C05481=1226.735,157.373,-52.424,-177.853,5.794,148.385
C05482=1226.731,157.623,-52.446,-177.851,5.795,148.384
C05483=1226.726,157.871,-52.468,-177.848,5.797,148.384
C05484=1226.721,158.120,-52.490,-177.846,5.798,148.383
C05485=1226.717,158.370,-52.511,-177.843,5.799,148.383
C05486=1226.712,158.619,-52.533,-177.841,5.800,148.382
C05487=1226.707,158.867,-52.555,-177.838,5.802,148.382
C05488=1226.703,159.117,-52.577,-177.836,5.803,148.381
C05489=1226.697,159.386,-52.600,-177.833,5.804,148.381
C05490=1226.693,159.655,-52.623,-177.830,5.806,148.380
C05491=1226.687,159.924,-52.647,-177.828,5.807,148.380
C05492=1226.683,160.193,-52.670,-177.824,5.808,148.379
C05493=1226.678,160.441,-52.691,-177.822,5.810,148.379
C05494=1226.674,160.691,-52.713,-177.820,5.811,148.379
C05495=1226.669,160.939,-52.735,-177.817,5.813,148.378
C05496=1226.664,161.189,-52.756,-177.814,5.814,148.378
C05497=1226.659,161.438,-52.778,-177.812,5.815,148.377
C05498=1226.654,161.687,-52.800,-177.809,5.816,148.377
C05499=1226.649,161.936,-52.822,-177.807,5.818,148.376
C05500=1226.644,162.185,-52.844,-177.804,5.819,148.376
C05501=1226.640,162.434,-52.866,-177.801,5.820,148.375
C05502=1226.635,162.683,-52.888,-177.799,5.821,148.375
C05503=1226.630,162.932,-52.909,-177.797,5.823,148.375
C05504=1226.626,163.181,-52.931,-177.794,5.824,148.374
C05505=1226.621,163.430,-52.953,-177.791,5.826,148.374
C05506=1226.617,163.679,-52.975,-177.789,5.828,148.373
C05507=1226.612,163.928,-52.997,-177.786,5.828,148.373
C05508=1226.608,164.177,-53.019,-177.783,5.830,148.372
C05509=1226.603,164.426,-53.040,-177.781,5.831,148.372
C05510=1226.599,164.675,-53.062,-177.778,5.833,148.371
C05511=1226.594,164.924,-53.084,-177.776,5.834,148.371
C05512=1226.590,165.173,-53.106,-177.773,5.835,148.370
C05513=1226.584,165.422,-53.129,-177.771,5.836,148.370
C05514=1226.579,165.670,-53.150,-177.768,5.838,148.369
C05515=1226.575,165.920,-53.172,-177.766,5.839,148.369
C05516=1226.570,166.168,-53.194,-177.763,5.840,148.368
C05517=1226.566,166.418,-53.216,-177.760,5.842,148.368
C05518=1226.561,166.666,-53.238,-177.758,5.843,148.368
C05519=1226.557,166.916,-53.260,-177.755,5.845,148.367
C05520=1226.551,167.165,-53.282,-177.753,5.846,148.367
C05521=1226.547,167.414,-53.304,-177.750,5.848,148.366
C05522=1226.542,167.663,-53.326,-177.748,5.848,148.366
C05523=1226.538,167.912,-53.348,-177.745,5.850,148.365
C05524=1226.534,168.161,-53.371,-177.742,5.852,148.365
C05525=1226.528,168.410,-53.393,-177.740,5.853,148.365
C05526=1226.524,168.659,-53.415,-177.737,5.854,148.364
C05527=1226.519,168.908,-53.437,-177.735,5.855,148.364
C05528=1226.515,169.157,-53.459,-177.732,5.857,148.363
C05529=1226.510,169.406,-53.480,-177.730,5.858,148.363
C05530=1226.505,169.655,-53.504,-177.727,5.860,148.362
C05531=1226.500,169.903,-53.525,-177.724,5.861,148.362
C05532=1226.496,170.153,-53.547,-177.722,5.862,148.361
C05533=1226.490,170.402,-53.570,-177.719,5.864,148.361
C05534=1226.486,170.651,-53.592,-177.717,5.865,148.361
C05535=1226.482,170.899,-53.614,-177.715,5.867,148.360
C05536=1226.477,171.148,-53.636,-177.712,5.867,148.360
C05537=1226.472,171.398,-53.659,-177.709,5.869,148.359
C05538=1226.467,171.647,-53.681,-177.707,5.871,148.359
C05539=1226.463,171.895,-53.703,-177.704,5.872,148.358
C05540=1226.458,172.144,-53.726,-177.701,5.874,148.358
C05541=1226.454,172.394,-53.748,-177.699,5.875,148.358
C05542=1226.449,172.642,-53.770,-177.697,5.876,148.357
C05543=1226.444,172.891,-53.793,-177.693,5.878,148.357
C05544=1226.440,173.141,-53.815,-177.691,5.879,148.356
C05545=1226.435,173.389,-53.837,-177.689,5.881,148.356
C05546=1226.430,173.638,-53.860,-177.687,5.882,148.356
C05547=1226.425,173.887,-53.881,-177.684,5.883,148.355
C05548=1226.421,174.136,-53.904,-177.681,5.885,148.355
C05549=1226.416,174.385,-53.927,-177.679,5.886,148.354
C05550=1226.412,174.633,-53.949,-177.676,5.888,148.354
C05551=1226.407,174.883,-53.971,-177.674,5.889,148.353
C05552=1226.402,175.132,-53.994,-177.671,5.890,148.353
C05553=1226.398,175.380,-54.016,-177.668,5.892,148.353
C05554=1226.393,175.630,-54.039,-177.666,5.893,148.352
C05555=1226.389,175.879,-54.062,-177.663,5.895,148.352
C05556=1226.384,176.127,-54.083,-177.660,5.897,148.351
C05557=1226.379,176.376,-54.107,-177.658,5.898,148.351
C05558=1226.375,176.626,-54.129,-177.655,5.899,148.350
C05559=1226.370,176.874,-54.152,-177.653,5.900,148.350
C05560=1226.366,177.123,-54.174,-177.650,5.902,148.349
C05561=1226.361,177.372,-54.197,-177.648,5.904,148.349
C05562=1226.356,177.621,-54.219,-177.645,5.905,148.349
C05563=1226.352,177.870,-54.242,-177.642,5.906,148.348
C05564=1226.347,178.119,-54.264,-177.640,5.908,148.348
C05565=1226.342,178.367,-54.287,-177.638,5.909,148.347
C05566=1226.337,178.617,-54.309,-177.635,5.911,148.347
C05567=1226.333,178.866,-54.332,-177.633,5.912,148.346
C05568=1226.328,179.115,-54.354,-177.630,5.914,148.346
C05569=1226.324,179.364,-54.377,-177.627,5.915,148.346
C05570=1226.319,179.613,-54.401,-177.625,5.916,148.345
C05571=1226.315,179.862,-54.423,-177.622,5.918,148.345
C05572=1226.310,180.110,-54.446,-177.619,5.920,148.344
C05573=1226.305,180.360,-54.468,-177.617,5.921,148.344
C05574=1226.301,180.609,-54.491,-177.615,5.923,148.344
C05575=1226.295,180.857,-54.514,-177.611,5.924,148.343
C05576=1226.291,181.106,-54.536,-177.609,5.925,148.343
C05577=1226.286,181.355,-54.559,-177.607,5.927,148.342
C05578=1226.282,181.604,-54.582,-177.604,5.929,148.342
C05579=1226.277,181.853,-54.604,-177.601,5.929,148.341
C05580=1226.273,182.102,-54.627,-177.599,5.931,148.341
C05581=1226.268,182.351,-54.651,-177.596,5.933,148.341
C05582=1226.263,182.600,-54.674,-177.594,5.934,148.340
C05583=1226.259,182.848,-54.696,-177.591,5.936,148.340
C05584=1226.254,183.097,-54.719,-177.589,5.937,148.339
C05585=1226.250,183.346,-54.742,-177.586,5.938,148.339
C05586=1226.245,183.595,-54.765,-177.584,5.940,148.339
C05587=1226.240,183.845,-54.788,-177.581,5.941,148.338
C05588=1226.236,184.093,-54.810,-177.578,5.943,148.338
C05589=1226.231,184.342,-54.833,-177.576,5.945,148.337
C05590=1226.226,184.591,-54.857,-177.574,5.946,148.337
C05591=1226.222,184.840,-54.880,-177.571,5.947,148.337
C05592=1226.217,185.089,-54.902,-177.568,5.949,148.336
C05593=1226.213,185.359,-54.927,-177.565,5.951,148.336
C05594=1226.208,185.628,-54.952,-177.563,5.953,148.335
C05595=1226.202,185.898,-54.977,-177.560,5.955,148.335
C05596=1226.198,186.167,-55.002,-177.557,5.955,148.334
C05597=1226.193,186.416,-55.025,-177.555,5.957,148.334
C05598=1226.187,186.665,-55.048,-177.552,5.959,148.334
C05599=1226.183,186.914,-55.071,-177.549,5.961,148.333
C05600=1226.179,187.163,-55.094,-177.547,5.961,148.333
C05601=1226.174,187.412,-55.117,-177.544,5.963,148.332
C05602=1226.169,187.661,-55.140,-177.542,5.965,148.332
C05603=1226.165,187.910,-55.163,-177.539,5.966,148.332
C05604=1226.161,188.159,-55.187,-177.537,5.968,148.331
C05605=1226.155,188.407,-55.210,-177.534,5.969,148.331
C05606=1226.151,188.656,-55.233,-177.532,5.970,148.330
C05607=1226.146,188.905,-55.256,-177.529,5.972,148.330
C05608=1226.142,189.154,-55.279,-177.526,5.974,148.330
C05609=1226.137,189.403,-55.302,-177.524,5.975,148.329
C05610=1226.133,189.652,-55.326,-177.522,5.977,148.329
C05611=1226.128,189.901,-55.349,-177.518,5.979,148.328
C05612=1226.124,190.150,-55.372,-177.516,5.980,148.328
C05613=1226.119,190.398,-55.395,-177.514,5.981,148.328
C05614=1226.114,190.647,-55.418,-177.511,5.983,148.327
C05615=1226.109,190.896,-55.442,-177.508,5.985,148.327
C05616=1226.105,191.145,-55.465,-177.506,5.986,148.327
C05617=1226.100,191.394,-55.488,-177.503,5.988,148.326
C05618=1226.096,191.643,-55.511,-177.501,5.989,148.326
C05619=1226.092,191.891,-55.535,-177.498,5.991,148.325
C05620=1226.087,192.140,-55.558,-177.496,5.992,148.325
C05621=1226.082,192.389,-55.582,-177.493,5.994,148.325
C05622=1226.077,192.638,-55.605,-177.491,5.996,148.324
C05623=1226.073,192.887,-55.629,-177.487,5.997,148.324
C05624=1226.068,193.136,-55.652,-177.485,5.999,148.323
C05625=1226.063,193.385,-55.675,-177.483,6.000,148.323
C05626=1226.060,193.634,-55.699,-177.480,6.002,148.323
C05627=1226.054,193.882,-55.722,-177.478,6.003,148.322
C05628=1226.050,194.131,-55.745,-177.475,6.005,148.322
C05629=1226.045,194.380,-55.768,-177.473,6.007,148.322
C05630=1226.040,194.629,-55.792,-177.470,6.008,148.321
C05631=1226.036,194.877,-55.816,-177.467,6.009,148.321
C05632=1226.031,195.126,-55.839,-177.465,6.011,148.320
C05633=1226.027,195.375,-55.863,-177.462,6.013,148.320
C05634=1226.022,195.624,-55.886,-177.460,6.015,148.320
C05635=1226.017,195.873,-55.910,-177.457,6.016,148.319
C05636=1226.013,196.122,-55.933,-177.455,6.018,148.319
C05637=1226.008,196.371,-55.957,-177.452,6.019,148.318
C05638=1226.003,196.620,-55.980,-177.449,6.021,148.318
C05639=1225.999,196.868,-56.004,-177.447,6.022,148.318
C05640=1225.994,197.117,-56.028,-177.444,6.024,148.317
C05641=1225.990,197.366,-56.051,-177.442,6.026,148.317
C05642=1225.985,197.615,-56.075,-177.439,6.028,148.317
C05643=1225.980,197.864,-56.098,-177.437,6.029,148.316
C05644=1225.976,198.113,-56.122,-177.434,6.031,148.316
C05645=1225.971,198.361,-56.146,-177.431,6.032,148.315
C05646=1225.967,198.610,-56.169,-177.429,6.034,148.315
C05647=1225.963,198.859,-56.194,-177.426,6.035,148.315
C05648=1225.958,199.109,-56.217,-177.424,6.037,148.314
C05649=1225.953,199.358,-56.240,-177.421,6.039,148.314
C05650=1225.949,199.606,-56.264,-177.419,6.041,148.313
C05651=1225.944,199.855,-56.288,-177.416,6.042,148.313
C05652=1225.940,200.103,-56.312,-177.414,6.043,148.313
C05653=1225.935,200.352,-56.335,-177.411,6.045,148.312
C05654=1225.930,200.601,-56.360,-177.408,6.047,148.312
C05655=1225.925,200.850,-56.383,-177.405,6.049,148.312
C05656=1225.921,201.099,-56.407,-177.403,6.050,148.311
C05657=1225.916,201.348,-56.431,-177.401,6.052,148.311
C05658=1225.912,201.596,-56.455,-177.398,6.053,148.310
C05659=1225.907,201.845,-56.478,-177.395,6.055,148.310
C05660=1225.903,202.094,-56.502,-177.393,6.057,148.310
C05661=1225.899,202.343,-56.526,-177.391,6.058,148.309
C05662=1225.894,202.592,-56.551,-177.388,6.060,148.309
C05663=1225.889,202.841,-56.574,-177.385,6.062,148.309
C05664=1225.885,203.089,-56.598,-177.383,6.064,148.308
C05665=1225.880,203.338,-56.622,-177.380,6.064,148.308
C05666=1225.875,203.587,-56.645,-177.378,6.066,148.307
C05667=1225.871,203.835,-56.669,-177.375,6.068,148.307
C05668=1225.866,204.085,-56.694,-177.372,6.070,148.307
C05669=1225.862,204.334,-56.718,-177.370,6.072,148.306
C05670=1225.857,204.582,-56.742,-177.368,6.073,148.306
C05671=1225.853,204.831,-56.765,-177.365,6.075,148.306
C05672=1225.848,205.080,-56.789,-177.362,6.076,148.305
C05673=1225.843,205.328,-56.814,-177.360,6.078,148.305
C05674=1225.839,205.577,-56.837,-177.357,6.080,148.305
C05675=1225.835,205.826,-56.862,-177.354,6.082,148.304
C05676=1225.830,206.075,-56.886,-177.352,6.083,148.304
C05677=1225.825,206.324,-56.910,-177.349,6.085,148.303
C05678=1225.820,206.573,-56.934,-177.347,6.086,148.303
C05679=1225.816,206.821,-56.958,-177.344,6.088,148.303
C05680=1225.812,207.070,-56.982,-177.341,6.090,148.302
C05681=1225.807,207.319,-57.006,-177.339,6.091,148.302
C05682=1225.802,207.568,-57.030,-177.337,6.093,148.302
C05683=1225.798,207.816,-57.055,-177.334,6.095,148.301
C05684=1225.793,208.065,-57.079,-177.331,6.097,148.301
C05685=1225.789,208.315,-57.103,-177.329,6.099,148.301
C05686=1225.784,208.563,-57.127,-177.326,6.100,148.300
C05687=1225.779,208.812,-57.152,-177.324,6.101,148.300
C05688=1225.775,209.060,-57.176,-177.321,6.103,148.300
C05689=1225.771,209.309,-57.200,-177.319,6.105,148.299
C05690=1225.766,209.558,-57.225,-177.316,6.107,148.299
C05691=1225.761,209.807,-57.248,-177.313,6.109,148.299
C05692=1225.757,210.056,-57.272,-177.311,6.111,148.298
C05693=1225.752,210.304,-57.297,-177.309,6.112,148.298
C05694=1225.748,210.553,-57.321,-177.306,6.114,148.298
C05695=1225.743,210.802,-57.346,-177.303,6.115,148.297
C05696=1225.738,211.051,-57.370,-177.300,6.117,148.297
C05697=1225.733,211.321,-57.397,-177.298,6.119,148.296
C05698=1225.728,211.592,-57.423,-177.295,6.121,148.296
C05699=1225.724,211.862,-57.449,-177.292,6.123,148.296
C05700=1225.719,212.132,-57.476,-177.290,6.124,148.295
C05701=1225.714,212.381,-57.501,-177.287,6.126,148.295
C05702=1225.710,212.630,-57.525,-177.285,6.128,148.295
C05703=1225.705,212.879,-57.550,-177.281,6.130,148.294
C05704=1225.700,213.127,-57.574,-177.279,6.132,148.294
C05705=1225.696,213.376,-57.598,-177.276,6.133,148.294
C05706=1225.692,213.625,-57.623,-177.274,6.135,148.293
C05707=1225.687,213.873,-57.647,-177.271,6.136,148.293
C05708=1225.682,214.122,-57.672,-177.269,6.138,148.293
C05709=1225.678,214.371,-57.696,-177.266,6.140,148.292
C05710=1225.673,214.620,-57.721,-177.264,6.142,148.292
C05711=1225.669,214.868,-57.745,-177.261,6.144,148.292
C05712=1225.664,215.118,-57.770,-177.258,6.146,148.291
C05713=1225.660,215.366,-57.794,-177.256,6.147,148.291
C05714=1225.655,215.615,-57.819,-177.254,6.148,148.290
C05715=1225.651,215.863,-57.844,-177.251,6.150,148.290
C05716=1225.646,216.112,-57.869,-177.248,6.152,148.290
C05717=1225.641,216.361,-57.893,-177.246,6.154,148.289
C05718=1225.637,216.610,-57.918,-177.243,6.156,148.289
C05719=1225.632,216.859,-57.942,-177.240,6.158,148.289
C05720=1225.628,217.108,-57.967,-177.238,6.160,148.289
C05721=1225.623,217.356,-57.992,-177.235,6.161,148.288
C05722=1225.619,217.604,-58.016,-177.233,6.163,148.288
C05723=1225.614,217.854,-58.041,-177.230,6.164,148.287
C05724=1225.609,218.103,-58.066,-177.228,6.166,148.287
C05725=1225.605,218.351,-58.090,-177.225,6.168,148.287
C05726=1225.601,218.600,-58.116,-177.223,6.170,148.286
C05727=1225.596,218.848,-58.140,-177.220,6.172,148.286
C05728=1225.592,219.098,-58.165,-177.217,6.174,148.286
C05729=1225.587,219.346,-58.190,-177.215,6.175,148.286
C05730=1225.582,219.594,-58.214,-177.212,6.177,148.285
C05731=1225.578,219.844,-58.239,-177.209,6.179,148.285
C05732=1225.573,220.092,-58.264,-177.207,6.180,148.284
C05733=1225.569,220.341,-58.289,-177.205,6.182,148.284
C05734=1225.564,220.589,-58.314,-177.202,6.184,148.284
C05735=1225.560,220.839,-58.339,-177.200,6.186,148.284
C05736=1225.556,221.087,-58.364,-177.197,6.188,148.283
C05737=1225.550,221.335,-58.388,-177.195,6.190,148.283
C05738=1225.546,221.585,-58.413,-177.192,6.192,148.283
C05739=1225.542,221.833,-58.438,-177.189,6.194,148.282
C05740=1225.537,222.082,-58.463,-177.187,6.195,148.282
C05741=1225.532,222.330,-58.489,-177.184,6.197,148.282
C05742=1225.529,222.579,-58.513,-177.182,6.198,148.281
C05743=1225.524,222.828,-58.538,-177.180,6.200,148.281
C05744=1225.519,223.077,-58.563,-177.177,6.202,148.281
C05745=1225.514,223.326,-58.588,-177.174,6.204,148.280
C05746=1225.511,223.574,-58.613,-177.172,6.206,148.280
C05747=1225.506,223.823,-58.638,-177.169,6.208,148.280
C05748=1225.501,224.072,-58.664,-177.166,6.210,148.279
C05749=1225.496,224.320,-58.688,-177.164,6.211,148.279
C05750=1225.492,224.569,-58.714,-177.161,6.213,148.279
C05751=1225.488,224.817,-58.738,-177.159,6.215,148.278
C05752=1225.483,225.066,-58.764,-177.156,6.217,148.278
C05753=1225.478,225.315,-58.789,-177.153,6.219,148.278
C05754=1225.474,225.564,-58.814,-177.151,6.220,148.277
C05755=1225.469,225.813,-58.839,-177.149,6.222,148.277
C05756=1225.465,226.061,-58.864,-177.146,6.224,148.277
C05757=1225.460,226.310,-58.889,-177.144,6.226,148.277
C05758=1225.456,226.559,-58.915,-177.141,6.228,148.276
C05759=1225.451,226.807,-58.940,-177.139,6.230,148.276
C05760=1225.447,227.056,-58.965,-177.136,6.231,148.276
C05761=1225.442,227.304,-58.990,-177.133,6.233,148.275
C05762=1225.438,227.553,-59.015,-177.131,6.235,148.275
C05763=1225.434,227.802,-59.041,-177.128,6.237,148.275
C05764=1225.429,228.050,-59.066,-177.125,6.239,148.274
C05765=1225.424,228.300,-59.091,-177.123,6.241,148.274
C05766=1225.420,228.548,-59.116,-177.120,6.243,148.274
C05767=1225.415,228.797,-59.142,-177.118,6.244,148.273
C05768=1225.410,229.045,-59.167,-177.116,6.246,148.273
C05769=1225.406,229.294,-59.193,-177.113,6.248,148.273
C05770=1225.402,229.543,-59.218,-177.111,6.250,148.273
C05771=1225.397,229.791,-59.244,-177.108,6.251,148.272
C05772=1225.393,230.040,-59.269,-177.105,6.253,148.272
C05773=1225.388,230.289,-59.294,-177.103,6.255,148.272
C05774=1225.384,230.537,-59.319,-177.100,6.257,148.271
C05775=1225.380,230.786,-59.345,-177.098,6.259,148.271
C05776=1225.375,231.035,-59.370,-177.095,6.261,148.271
C05777=1225.371,231.283,-59.395,-177.093,6.263,148.271
C05778=1225.366,231.531,-59.421,-177.090,6.265,148.270
C05779=1225.362,231.780,-59.447,-177.088,6.267,148.270
C05780=1225.357,232.029,-59.472,-177.085,6.269,148.270
C05781=1225.352,232.278,-59.497,-177.082,6.270,148.269
C05782=1225.348,232.527,-59.523,-177.080,6.272,148.269
C05783=1225.344,232.775,-59.549,-177.077,6.274,148.269
C05784=1225.339,233.024,-59.574,-177.075,6.276,148.268
C05785=1225.334,233.273,-59.600,-177.073,6.277,148.268
C05786=1225.330,233.521,-59.626,-177.070,6.279,148.268
C05787=1225.325,233.770,-59.651,-177.068,6.281,148.268
C05788=1225.321,234.018,-59.677,-177.065,6.283,148.267
C05789=1225.316,234.267,-59.703,-177.062,6.285,148.267
C05790=1225.311,234.516,-59.728,-177.060,6.287,148.267
C05791=1225.307,234.765,-59.753,-177.057,6.289,148.266
C05792=1225.303,235.013,-59.779,-177.055,6.290,148.266
C05793=1225.298,235.262,-59.804,-177.052,6.293,148.266
C05794=1225.294,235.510,-59.830,-177.050,6.295,148.266
C05795=1225.290,235.759,-59.856,-177.047,6.296,148.265
C05796=1225.285,236.007,-59.881,-177.045,6.298,148.265
C05797=1225.280,236.256,-59.908,-177.042,6.300,148.265
C05798=1225.276,236.505,-59.933,-177.039,6.302,148.264
C05799=1225.271,236.754,-59.959,-177.037,6.304,148.264
C05800=1225.267,237.002,-59.985,-177.035,6.306,148.264
C05801=1225.262,237.273,-60.013,-177.032,6.308,148.264
C05802=1225.257,237.545,-60.041,-177.029,6.310,148.263
C05803=1225.252,237.816,-60.069,-177.026,6.313,148.263
C05804=1225.248,238.088,-60.098,-177.024,6.314,148.263
C05805=1225.243,238.336,-60.123,-177.021,6.316,148.262
C05806=1225.238,238.585,-60.150,-177.018,6.318,148.262
C05807=1225.234,238.834,-60.175,-177.016,6.320,148.262
C05808=1225.230,239.083,-60.201,-177.013,6.322,148.261
C05809=1225.225,239.331,-60.226,-177.011,6.324,148.261
C05810=1225.220,239.580,-60.252,-177.008,6.326,148.261
C05811=1225.216,239.828,-60.279,-177.006,6.328,148.261
C05812=1225.212,240.077,-60.305,-177.003,6.330,148.260
C05813=1225.207,240.326,-60.331,-177.000,6.332,148.260
C05814=1225.203,240.574,-60.356,-176.998,6.333,148.260
C05815=1225.198,240.823,-60.382,-176.996,6.336,148.260
C05816=1225.194,241.071,-60.409,-176.993,6.338,148.259
C05817=1225.189,241.320,-60.435,-176.991,6.339,148.259
C05818=1225.185,241.568,-60.460,-176.988,6.341,148.259
C05819=1225.180,241.817,-60.486,-176.985,6.343,148.258
C05820=1225.176,242.065,-60.513,-176.983,6.345,148.258
C05821=1225.172,242.314,-60.539,-176.981,6.347,148.258
C05822=1225.167,242.563,-60.565,-176.978,6.349,148.258
C05823=1225.162,242.812,-60.591,-176.975,6.351,148.257
C05824=1225.158,243.059,-60.617,-176.973,6.353,148.257
C05825=1225.153,243.309,-60.643,-176.971,6.355,148.257
C05826=1225.149,243.557,-60.669,-176.968,6.357,148.257
C05827=1225.145,243.806,-60.695,-176.965,6.359,148.256
C05828=1225.140,244.055,-60.722,-176.963,6.361,148.256
C05829=1225.136,244.303,-60.747,-176.961,6.363,148.256
C05830=1225.131,244.551,-60.774,-176.958,6.365,148.256
C05831=1225.126,244.800,-60.800,-176.955,6.367,148.255
C05832=1225.122,245.048,-60.826,-176.953,6.369,148.255
C05833=1225.118,245.297,-60.852,-176.950,6.370,148.255
C05834=1225.113,245.546,-60.878,-176.948,6.373,148.255
C05835=1225.109,245.794,-60.905,-176.945,6.374,148.254
C05836=1225.104,246.043,-60.931,-176.943,6.376,148.254
C05837=1225.100,246.292,-60.958,-176.940,6.378,148.254
C05838=1225.095,246.540,-60.984,-176.938,6.380,148.254
C05839=1225.091,246.788,-61.010,-176.935,6.382,148.253
C05840=1225.086,247.037,-61.036,-176.933,6.384,148.253
C05841=1225.082,247.286,-61.063,-176.930,6.386,148.253
C05842=1225.078,247.534,-61.089,-176.928,6.388,148.253
C05843=1225.073,247.783,-61.116,-176.925,6.390,148.252
C05844=1225.069,248.032,-61.142,-176.923,6.392,148.252
C05845=1225.064,248.280,-61.169,-176.920,6.394,148.252
C05846=1225.060,248.529,-61.194,-176.918,6.396,148.252
C05847=1225.055,248.777,-61.221,-176.915,6.398,148.251
C05848=1225.051,249.026,-61.247,-176.913,6.400,148.251
C05849=1225.046,249.275,-61.274,-176.910,6.402,148.251
C05850=1225.042,249.523,-61.301,-176.908,6.405,148.251
C05851=1225.037,249.771,-61.327,-176.905,6.407,148.250
C05852=1225.033,250.020,-61.353,-176.902,6.408,148.250
C05853=1225.028,250.268,-61.380,-176.900,6.410,148.250
C05854=1225.024,250.517,-61.406,-176.898,6.413,148.250
C05855=1225.019,250.765,-61.433,-176.895,6.414,148.249
C05856=1225.015,251.014,-61.459,-176.892,6.416,148.249
C05857=1225.010,251.263,-61.486,-176.890,6.419,148.249
C05858=1225.006,251.511,-61.513,-176.888,6.420,148.249
C05859=1225.002,251.759,-61.539,-176.885,6.422,148.248
C05860=1224.997,252.008,-61.566,-176.882,6.424,148.248
C05861=1224.993,252.257,-61.592,-176.880,6.426,148.248
C05862=1224.988,252.505,-61.619,-176.878,6.428,148.248
C05863=1224.984,252.754,-61.645,-176.875,6.430,148.247
C05864=1224.979,253.002,-61.672,-176.873,6.432,148.247
C05865=1224.975,253.251,-61.699,-176.870,6.434,148.247
C05866=1224.971,253.499,-61.726,-176.868,6.436,148.247
C05867=1224.966,253.748,-61.752,-176.865,6.439,148.246
C05868=1224.961,253.997,-61.779,-176.862,6.441,148.246
C05869=1224.957,254.245,-61.805,-176.860,6.443,148.246
C05870=1224.953,254.493,-61.833,-176.857,6.445,148.246
C05871=1224.948,254.742,-61.860,-176.855,6.447,148.246
C05872=1224.944,254.990,-61.886,-176.852,6.449,148.245
C05873=1224.940,255.240,-61.913,-176.850,6.451,148.245
C05874=1224.935,255.488,-61.940,-176.848,6.453,148.245
C05875=1224.931,255.737,-61.966,-176.845,6.455,148.245
C05876=1224.926,255.985,-61.993,-176.842,6.457,148.244
C05877=1224.922,256.234,-62.020,-176.840,6.459,148.244
C05878=1224.918,256.482,-62.047,-176.838,6.461,148.244
C05879=1224.913,256.730,-62.074,-176.835,6.463,148.244
C05880=1224.909,256.979,-62.101,-176.832,6.466,148.244
C05881=1224.904,257.227,-62.128,-176.830,6.468,148.243
C05882=1224.900,257.475,-62.155,-176.827,6.469,148.243
C05883=1224.895,257.724,-62.182,-176.825,6.472,148.243
C05884=1224.891,257.972,-62.209,-176.822,6.474,148.243
C05885=1224.886,258.222,-62.235,-176.820,6.475,148.242
C05886=1224.882,258.470,-62.262,-176.818,6.478,148.242
C05887=1224.878,258.718,-62.290,-176.815,6.479,148.242
C05888=1224.873,258.967,-62.317,-176.813,6.481,148.242
C05889=1224.869,259.215,-62.344,-176.810,6.484,148.241
C05890=1224.864,259.464,-62.371,-176.807,6.486,148.241
C05891=1224.860,259.712,-62.397,-176.805,6.488,148.241
C05892=1224.856,259.960,-62.424,-176.803,6.490,148.241
C05893=1224.851,260.209,-62.451,-176.800,6.492,148.240
C05894=1224.847,260.458,-62.479,-176.797,6.494,148.240
C05895=1224.842,260.707,-62.506,-176.795,6.496,148.240
C05896=1224.838,260.955,-62.533,-176.793,6.498,148.240
C05897=1224.834,261.203,-62.559,-176.790,6.500,148.240
C05898=1224.829,261.452,-62.586,-176.788,6.502,148.239
C05899=1224.824,261.700,-62.614,-176.785,6.505,148.239
C05900=1224.821,261.949,-62.642,-176.783,6.507,148.239
C05901=1224.816,262.197,-62.669,-176.780,6.509,148.239
C05902=1224.811,262.446,-62.696,-176.777,6.511,148.238
C05903=1224.807,262.694,-62.723,-176.775,6.513,148.238
C05904=1224.802,262.943,-62.750,-176.773,6.515,148.238
C05905=1224.797,263.215,-62.780,-176.769,6.518,148.238
C05906=1224.792,263.488,-62.810,-176.767,6.520,148.238
C05907=1224.788,263.761,-62.840,-176.764,6.523,148.238
C05908=1224.784,264.033,-62.870,-176.762,6.525,148.237
C05909=1224.779,264.282,-62.897,-176.759,6.527,148.237
C05910=1224.774,264.530,-62.924,-176.757,6.529,148.237
C05911=1224.770,264.779,-62.951,-176.754,6.531,148.237
C05912=1224.766,265.027,-62.979,-176.752,6.533,148.236
C05913=1224.761,265.276,-63.006,-176.749,6.536,148.236
C05914=1224.757,265.524,-63.033,-176.747,6.538,148.236
C05915=1224.752,265.772,-63.061,-176.744,6.540,148.236
C05916=1224.748,266.021,-63.088,-176.742,6.542,148.236
C05917=1224.744,266.270,-63.115,-176.740,6.544,148.235
C05918=1224.739,266.518,-63.143,-176.737,6.546,148.235
C05919=1224.735,266.766,-63.170,-176.734,6.549,148.235
C05920=1224.731,267.015,-63.198,-176.732,6.551,148.235
C05921=1224.726,267.263,-63.226,-176.730,6.553,148.235
C05922=1224.721,267.512,-63.253,-176.727,6.555,148.234
C05923=1224.716,267.760,-63.281,-176.724,6.557,148.234
C05924=1224.712,268.009,-63.308,-176.722,6.559,148.234
C05925=1224.708,268.257,-63.336,-176.720,6.561,148.234
C05926=1224.703,268.505,-63.363,-176.717,6.564,148.234
C05927=1224.699,268.754,-63.390,-176.714,6.566,148.233
C05928=1224.695,269.002,-63.418,-176.712,6.568,148.233
C05929=1224.690,269.251,-63.445,-176.710,6.570,148.233
C05930=1224.686,269.499,-63.473,-176.707,6.572,148.233
C05931=1224.682,269.748,-63.501,-176.705,6.574,148.233
C05932=1224.678,269.996,-63.528,-176.702,6.577,148.233
C05933=1224.672,270.245,-63.556,-176.700,6.579,148.232
C05934=1224.668,270.493,-63.584,-176.697,6.581,148.232
C05935=1224.664,270.741,-63.612,-176.695,6.583,148.232
C05936=1224.659,270.990,-63.639,-176.692,6.585,148.232
C05937=1224.656,271.238,-63.667,-176.690,6.587,148.232
C05938=1224.651,271.487,-63.694,-176.687,6.590,148.231
C05939=1224.647,271.735,-63.722,-176.685,6.592,148.231
C05940=1224.642,271.984,-63.751,-176.682,6.594,148.231
C05941=1224.637,272.232,-63.778,-176.680,6.596,148.231
C05942=1224.633,272.480,-63.806,-176.678,6.598,148.231
C05943=1224.629,272.729,-63.833,-176.675,6.601,148.231
C05944=1224.625,272.977,-63.861,-176.672,6.603,148.230
C05945=1224.620,273.225,-63.889,-176.670,6.605,148.230
C05946=1224.616,273.474,-63.917,-176.668,6.607,148.230
C05947=1224.611,273.722,-63.944,-176.665,6.609,148.230
C05948=1224.607,273.971,-63.973,-176.662,6.612,148.230
C05949=1224.602,274.219,-64.001,-176.660,6.614,148.230
C05950=1224.598,274.467,-64.028,-176.658,6.616,148.229
C05951=1224.594,274.716,-64.056,-176.655,6.618,148.229
C05952=1224.590,274.964,-64.084,-176.653,6.620,148.229
C05953=1224.585,275.213,-64.112,-176.650,6.623,148.229
C05954=1224.580,275.461,-64.140,-176.648,6.625,148.229
C05955=1224.576,275.709,-64.168,-176.645,6.627,148.229
C05956=1224.572,275.958,-64.196,-176.643,6.629,148.228
C05957=1224.567,276.206,-64.224,-176.641,6.631,148.228
C05958=1224.563,276.455,-64.251,-176.638,6.634,148.228
C05959=1224.559,276.703,-64.279,-176.635,6.636,148.228
C05960=1224.554,276.952,-64.308,-176.633,6.638,148.228
C05961=1224.550,277.200,-64.336,-176.631,6.640,148.227
C05962=1224.546,277.448,-64.364,-176.629,6.642,148.227
C05963=1224.541,277.697,-64.392,-176.625,6.645,148.227
C05964=1224.537,277.944,-64.420,-176.623,6.647,148.227
C05965=1224.533,278.194,-64.447,-176.621,6.649,148.227
C05966=1224.528,278.442,-64.476,-176.619,6.651,148.227
C05967=1224.524,278.690,-64.504,-176.615,6.654,148.226
C05968=1224.519,278.939,-64.532,-176.613,6.656,148.226
C05969=1224.515,279.187,-64.561,-176.611,6.659,148.226
C05970=1224.511,279.435,-64.588,-176.609,6.660,148.226
C05971=1224.506,279.684,-64.617,-176.607,6.663,148.226
C05972=1224.502,279.932,-64.645,-176.603,6.665,148.226
C05973=1224.497,280.181,-64.674,-176.601,6.668,148.226
C05974=1224.493,280.429,-64.701,-176.599,6.670,148.225
C05975=1224.489,280.677,-64.730,-176.597,6.672,148.225
C05976=1224.484,280.925,-64.758,-176.594,6.675,148.225
C05977=1224.481,281.174,-64.786,-176.591,6.677,148.225
C05978=1224.475,281.422,-64.814,-176.589,6.679,148.225
C05979=1224.472,281.671,-64.842,-176.587,6.681,148.225
C05980=1224.467,281.920,-64.871,-176.584,6.684,148.225
C05981=1224.463,282.167,-64.899,-176.582,6.686,148.225
C05982=1224.458,282.416,-64.928,-176.579,6.688,148.224
C05983=1224.454,282.664,-64.956,-176.577,6.690,148.224
C05984=1224.450,282.912,-64.985,-176.574,6.693,148.224
C05985=1224.445,283.160,-65.013,-176.572,6.695,148.224
C05986=1224.441,283.409,-65.041,-176.570,6.697,148.224
C05987=1224.437,283.657,-65.069,-176.567,6.699,148.224
C05988=1224.432,283.906,-65.098,-176.564,6.702,148.224
C05989=1224.428,284.154,-65.126,-176.562,6.704,148.223
C05990=1224.424,284.402,-65.155,-176.560,6.706,148.223
C05991=1224.419,284.651,-65.184,-176.558,6.709,148.223
C05992=1224.415,284.899,-65.212,-176.554,6.711,148.223
C05993=1224.410,285.148,-65.240,-176.552,6.714,148.223
C05994=1224.406,285.396,-65.268,-176.550,6.716,148.223
C05995=1224.402,285.644,-65.298,-176.548,6.718,148.222
C05996=1224.397,285.893,-65.326,-176.545,6.721,148.222
C05997=1224.393,286.141,-65.354,-176.543,6.723,148.222
C05998=1224.388,286.390,-65.383,-176.540,6.725,148.222
C05999=1224.384,286.637,-65.411,-176.538,6.727,148.222
C06000=1224.380,286.886,-65.440,-176.535,6.730,148.222
C06001=1224.375,287.135,-65.469,-176.533,6.732,148.222
C06002=1224.371,287.382,-65.497,-176.531,6.734,148.222
C06003=1224.367,287.631,-65.526,-176.529,6.736,148.222
C06004=1224.362,287.880,-65.555,-176.525,6.739,148.221
C06005=1224.358,288.127,-65.583,-176.523,6.741,148.221
C06006=1224.354,288.376,-65.612,-176.521,6.743,148.221
C06007=1224.349,288.624,-65.641,-176.518,6.746,148.221
C06008=1224.345,288.872,-65.669,-176.516,6.748,148.221
C06009=1224.341,289.146,-65.701,-176.514,6.751,148.221
C06010=1224.336,289.421,-65.733,-176.511,6.753,148.221
C06011=1224.331,289.695,-65.764,-176.508,6.756,148.221
C06012=1224.326,289.969,-65.797,-176.505,6.758,148.220
C06013=1224.321,290.217,-65.825,-176.503,6.761,148.220
C06014=1224.317,290.465,-65.854,-176.501,6.764,148.220
C06015=1224.313,290.714,-65.883,-176.499,6.766,148.220
C06016=1224.309,290.961,-65.912,-176.496,6.768,148.220
C06017=1224.304,291.210,-65.940,-176.493,6.771,148.220
C06018=1224.300,291.458,-65.970,-176.491,6.773,148.220
C06019=1224.296,291.706,-65.998,-176.489,6.775,148.220
C06020=1224.291,291.955,-66.027,-176.486,6.778,148.220
C06021=1224.287,292.204,-66.056,-176.484,6.780,148.219
C06022=1224.283,292.452,-66.085,-176.482,6.782,148.219
C06023=1224.278,292.700,-66.114,-176.479,6.785,148.219
C06024=1224.274,292.948,-66.143,-176.476,6.787,148.219
C06025=1224.270,293.197,-66.171,-176.474,6.790,148.219
C06026=1224.266,293.445,-66.201,-176.472,6.792,148.219
C06027=1224.261,293.693,-66.230,-176.470,6.795,148.219
C06028=1224.256,293.942,-66.259,-176.467,6.797,148.219
C06029=1224.252,294.190,-66.288,-176.465,6.799,148.219
C06030=1224.249,294.438,-66.317,-176.462,6.802,148.219
C06031=1224.244,294.686,-66.345,-176.460,6.804,148.219
C06032=1224.239,294.934,-66.375,-176.458,6.806,148.218
C06033=1224.235,295.182,-66.404,-176.455,6.809,148.218
C06034=1224.231,295.431,-66.433,-176.453,6.811,148.218
C06035=1224.226,295.679,-66.462,-176.451,6.814,148.218
C06036=1224.222,295.927,-66.491,-176.449,6.816,148.218
C06037=1224.217,296.176,-66.520,-176.445,6.818,148.218
C06038=1224.214,296.424,-66.549,-176.443,6.821,148.218
C06039=1224.210,296.672,-66.578,-176.441,6.823,148.218
C06040=1224.205,296.920,-66.608,-176.438,6.826,148.218
C06041=1224.200,297.169,-66.636,-176.436,6.828,148.218
C06042=1224.196,297.417,-66.666,-176.434,6.830,148.217
C06043=1224.192,297.665,-66.695,-176.431,6.833,148.217
C06044=1224.188,297.914,-66.725,-176.429,6.835,148.217
C06045=1224.184,298.162,-66.754,-176.427,6.838,148.217
C06046=1224.179,298.410,-66.782,-176.424,6.841,148.217
C06047=1224.174,298.658,-66.812,-176.422,6.843,148.217
C06048=1224.170,298.907,-66.841,-176.420,6.845,148.217
C06049=1224.166,299.155,-66.871,-176.417,6.848,148.217
C06050=1224.162,299.403,-66.900,-176.415,6.850,148.217
C06051=1224.158,299.651,-66.930,-176.413,6.852,148.217
C06052=1224.153,299.899,-66.959,-176.410,6.855,148.217
C06053=1224.149,300.147,-66.988,-176.408,6.857,148.217
C06054=1224.144,300.395,-67.018,-176.406,6.860,148.217
C06055=1224.140,300.644,-67.046,-176.403,6.863,148.217
C06056=1224.136,300.893,-67.076,-176.401,6.865,148.216
C06057=1224.132,301.141,-67.105,-176.398,6.867,148.216
C06058=1224.127,301.389,-67.135,-176.396,6.870,148.216
C06059=1224.123,301.637,-67.164,-176.394,6.872,148.216
C06060=1224.118,301.885,-67.193,-176.392,6.874,148.216
C06061=1224.114,302.134,-67.223,-176.389,6.877,148.216
C06062=1224.109,302.382,-67.253,-176.387,6.880,148.216
C06063=1224.105,302.630,-67.282,-176.385,6.882,148.216
C06064=1224.101,302.878,-67.312,-176.382,6.885,148.216
C06065=1224.097,303.127,-67.341,-176.380,6.887,148.216
C06066=1224.093,303.375,-67.371,-176.377,6.889,148.216
C06067=1224.089,303.623,-67.401,-176.375,6.892,148.216
C06068=1224.085,303.871,-67.430,-176.372,6.894,148.216
C06069=1224.080,304.119,-67.460,-176.370,6.896,148.216
C06070=1224.076,304.368,-67.490,-176.368,6.900,148.216
C06071=1224.071,304.616,-67.519,-176.366,6.902,148.216
C06072=1224.067,304.864,-67.549,-176.364,6.904,148.215
C06073=1224.062,305.112,-67.578,-176.361,6.907,148.215
C06074=1224.058,305.360,-67.607,-176.359,6.909,148.215
C06075=1224.054,305.608,-67.638,-176.357,6.911,148.215
C06076=1224.049,305.856,-67.667,-176.354,6.914,148.215
C06077=1224.045,306.105,-67.697,-176.352,6.917,148.215
C06078=1224.041,306.353,-67.726,-176.350,6.919,148.215
C06079=1224.036,306.601,-67.756,-176.347,6.922,148.215
C06080=1224.032,306.849,-67.787,-176.345,6.924,148.215
C06081=1224.028,307.097,-67.816,-176.342,6.927,148.215
C06082=1224.024,307.346,-67.846,-176.340,6.929,148.215
C06083=1224.020,307.594,-67.875,-176.338,6.932,148.215
C06084=1224.015,307.842,-67.906,-176.335,6.935,148.215
C06085=1224.011,308.090,-67.935,-176.333,6.937,148.215
C06086=1224.007,308.338,-67.965,-176.331,6.939,148.215
C06087=1224.002,308.587,-67.995,-176.329,6.942,148.215
C06088=1223.998,308.835,-68.025,-176.326,6.944,148.215
C06089=1223.994,309.083,-68.054,-176.324,6.947,148.215
C06090=1223.990,309.331,-68.084,-176.322,6.950,148.215
C06091=1223.985,309.579,-68.115,-176.320,6.952,148.215
C06092=1223.981,309.827,-68.144,-176.317,6.954,148.215
C06093=1223.977,310.076,-68.173,-176.315,6.957,148.215
C06094=1223.972,310.323,-68.204,-176.313,6.959,148.215
C06095=1223.968,310.572,-68.234,-176.310,6.962,148.215
C06096=1223.964,310.819,-68.264,-176.308,6.965,148.215
C06097=1223.960,311.069,-68.294,-176.306,6.967,148.215
C06098=1223.955,311.317,-68.324,-176.303,6.970,148.215
C06099=1223.951,311.565,-68.354,-176.301,6.972,148.215
C06100=1223.947,311.813,-68.384,-176.299,6.974,148.214
C06101=1223.943,312.061,-68.414,-176.297,6.978,148.215
C06102=1223.938,312.309,-68.444,-176.295,6.980,148.215
C06103=1223.934,312.557,-68.474,-176.293,6.982,148.215
C06104=1223.929,312.806,-68.504,-176.290,6.985,148.215
C06105=1223.925,313.053,-68.535,-176.288,6.987,148.215
C06106=1223.921,313.302,-68.564,-176.285,6.990,148.215
C06107=1223.916,313.550,-68.595,-176.283,6.993,148.214
C06108=1223.912,313.798,-68.624,-176.281,6.995,148.214
C06109=1223.908,314.046,-68.655,-176.278,6.998,148.214
C06110=1223.904,314.295,-68.685,-176.277,7.000,148.215
C06111=1223.899,314.543,-68.716,-176.275,7.003,148.215
C06112=1223.895,314.790,-68.746,-176.272,7.006,148.215
C06113=1223.890,315.067,-68.779,-176.269,7.009,148.215
C06114=1223.886,315.342,-68.813,-176.267,7.011,148.215
C06115=1223.881,315.618,-68.846,-176.264,7.014,148.215
C06116=1223.877,315.893,-68.880,-176.262,7.017,148.215
C06117=1223.872,316.142,-68.910,-176.260,7.019,148.214
C06118=1223.868,316.390,-68.940,-176.257,7.022,148.214
C06119=1223.864,316.638,-68.971,-176.255,7.025,148.215
C06120=1223.859,316.887,-69.001,-176.253,7.027,148.215
C06121=1223.855,317.134,-69.031,-176.251,7.030,148.215
C06122=1223.850,317.382,-69.062,-176.249,7.032,148.215
C06123=1223.847,317.630,-69.092,-176.246,7.035,148.214
C06124=1223.842,317.879,-69.122,-176.244,7.038,148.214
C06125=1223.838,318.127,-69.153,-176.242,7.040,148.215
C06126=1223.834,318.375,-69.184,-176.239,7.043,148.215
C06127=1223.830,318.623,-69.214,-176.237,7.046,148.215
C06128=1223.825,318.871,-69.244,-176.235,7.048,148.215
C06129=1223.820,319.119,-69.275,-176.233,7.051,148.215
C06130=1223.817,319.368,-69.305,-176.231,7.053,148.215
C06131=1223.812,319.615,-69.336,-176.229,7.056,148.215
C06132=1223.809,319.863,-69.366,-176.226,7.059,148.215
C06133=1223.804,320.112,-69.396,-176.224,7.061,148.215
C06134=1223.800,320.360,-69.427,-176.222,7.064,148.215
C06135=1223.796,320.608,-69.457,-176.220,7.066,148.215
C06136=1223.791,320.856,-69.488,-176.218,7.069,148.215
C06137=1223.787,321.104,-69.519,-176.216,7.072,148.215
C06138=1223.783,321.352,-69.549,-176.213,7.074,148.215
C06139=1223.779,321.600,-69.580,-176.211,7.076,148.215
C06140=1223.774,321.848,-69.611,-176.209,7.079,148.215
C06141=1223.770,322.096,-69.641,-176.207,7.082,148.215
C06142=1223.766,322.345,-69.672,-176.204,7.085,148.215
C06143=1223.761,322.593,-69.702,-176.202,7.087,148.215
C06144=1223.757,322.841,-69.733,-176.201,7.090,148.215
C06145=1223.753,323.089,-69.763,-176.198,7.093,148.215
C06146=1223.749,323.337,-69.794,-176.196,7.095,148.215
C06147=1223.745,323.585,-69.825,-176.194,7.098,148.215
C06148=1223.740,323.833,-69.855,-176.192,7.101,148.215
C06149=1223.736,324.081,-69.886,-176.189,7.103,148.215
C06150=1223.732,324.330,-69.917,-176.187,7.106,148.216
C06151=1223.728,324.577,-69.947,-176.185,7.108,148.215
C06152=1223.723,324.825,-69.978,-176.183,7.111,148.215
C06153=1223.719,325.073,-70.010,-176.181,7.114,148.216
C06154=1223.715,325.321,-70.041,-176.179,7.116,148.216
C06155=1223.710,325.569,-70.072,-176.176,7.119,148.216
C06156=1223.707,325.817,-70.102,-176.174,7.122,148.216
C06157=1223.702,326.065,-70.133,-176.172,7.124,148.216
C06158=1223.698,326.313,-70.164,-176.170,7.127,148.216
C06159=1223.694,326.562,-70.195,-176.168,7.130,148.216
C06160=1223.689,326.810,-70.226,-176.166,7.132,148.216
C06161=1223.685,327.058,-70.256,-176.164,7.135,148.216
C06162=1223.681,327.306,-70.288,-176.162,7.137,148.216
C06163=1223.677,327.554,-70.318,-176.160,7.141,148.216
C06164=1223.672,327.802,-70.349,-176.157,7.143,148.216
C06165=1223.668,328.050,-70.380,-176.155,7.145,148.216
C06166=1223.664,328.298,-70.411,-176.153,7.149,148.216
C06167=1223.660,328.545,-70.442,-176.151,7.151,148.216
C06168=1223.656,328.794,-70.473,-176.149,7.153,148.217
C06169=1223.651,329.042,-70.504,-176.147,7.156,148.217
C06170=1223.647,329.291,-70.535,-176.145,7.159,148.217
C06171=1223.643,329.538,-70.566,-176.142,7.162,148.217
C06172=1223.638,329.786,-70.597,-176.141,7.165,148.217
C06173=1223.634,330.034,-70.628,-176.139,7.167,148.217
C06174=1223.630,330.282,-70.659,-176.136,7.170,148.217
C06175=1223.626,330.530,-70.691,-176.134,7.172,148.217
C06176=1223.622,330.778,-70.722,-176.132,7.175,148.217
C06177=1223.617,331.026,-70.752,-176.130,7.178,148.217
C06178=1223.613,331.274,-70.784,-176.128,7.180,148.217
C06179=1223.609,331.522,-70.815,-176.126,7.183,148.217
C06180=1223.605,331.771,-70.846,-176.124,7.186,148.218
C06181=1223.601,332.018,-70.877,-176.122,7.188,148.218
C06182=1223.596,332.266,-70.908,-176.120,7.192,148.218
C06183=1223.593,332.514,-70.940,-176.118,7.194,148.218
C06184=1223.588,332.762,-70.970,-176.116,7.196,148.218
C06185=1223.584,333.011,-71.002,-176.114,7.199,148.218
C06186=1223.580,333.258,-71.033,-176.112,7.202,148.218
C06187=1223.576,333.507,-71.064,-176.109,7.205,148.218
C06188=1223.571,333.754,-71.096,-176.108,7.208,148.218
C06189=1223.567,334.003,-71.127,-176.106,7.210,148.218
C06190=1223.562,334.250,-71.159,-176.103,7.213,148.218
C06191=1223.558,334.499,-71.190,-176.102,7.216,148.219
C06192=1223.554,334.746,-71.221,-176.100,7.218,148.219
C06193=1223.549,334.994,-71.252,-176.097,7.221,148.219
C06194=1223.546,335.242,-71.284,-176.095,7.223,148.219
C06195=1223.541,335.490,-71.315,-176.093,7.227,148.219
C06196=1223.537,335.738,-71.347,-176.092,7.229,148.219
C06197=1223.533,335.986,-71.377,-176.089,7.232,148.219
C06198=1223.529,336.234,-71.409,-176.087,7.235,148.219
C06199=1223.525,336.482,-71.441,-176.086,7.237,148.220
C06200=1223.521,336.730,-71.472,-176.083,7.240,148.220
C06201=1223.516,336.978,-71.503,-176.081,7.243,148.220
C06202=1223.512,337.227,-71.535,-176.080,7.246,148.220
C06203=1223.508,337.475,-71.567,-176.078,7.248,148.220
C06204=1223.504,337.722,-71.598,-176.075,7.251,148.220
C06205=1223.500,337.971,-71.630,-176.074,7.254,148.220
C06206=1223.495,338.218,-71.661,-176.071,7.257,148.220
C06207=1223.492,338.466,-71.693,-176.069,7.259,148.221
C06208=1223.487,338.714,-71.724,-176.068,7.262,148.221
C06209=1223.483,338.962,-71.756,-176.065,7.265,148.221
C06210=1223.478,339.210,-71.788,-176.064,7.267,148.221
C06211=1223.474,339.458,-71.819,-176.062,7.270,148.221
C06212=1223.470,339.706,-71.850,-176.060,7.273,148.221
C06213=1223.466,339.954,-71.882,-176.058,7.275,148.221
C06214=1223.462,340.202,-71.914,-176.056,7.278,148.221
C06215=1223.457,340.450,-71.945,-176.054,7.281,148.222
C06216=1223.454,340.698,-71.977,-176.052,7.284,148.222
C06217=1223.449,340.976,-72.013,-176.050,7.287,148.222
C06218=1223.443,341.253,-72.048,-176.047,7.290,148.222
C06219=1223.439,341.531,-72.083,-176.046,7.293,148.222
C06220=1223.435,341.808,-72.119,-176.043,7.296,148.222
C06221=1223.431,342.056,-72.151,-176.041,7.298,148.222
C06222=1223.426,342.305,-72.182,-176.039,7.302,148.223
C06223=1223.422,342.553,-72.214,-176.038,7.304,148.223
C06224=1223.418,342.801,-72.246,-176.036,7.307,148.223
C06225=1223.413,343.048,-72.278,-176.034,7.310,148.223
C06226=1223.409,343.296,-72.310,-176.032,7.312,148.223
C06227=1223.405,343.544,-72.341,-176.030,7.315,148.223
C06228=1223.401,343.792,-72.373,-176.028,7.318,148.224
C06229=1223.397,344.041,-72.405,-176.026,7.321,148.224
C06230=1223.392,344.288,-72.436,-176.025,7.323,148.224
C06231=1223.389,344.536,-72.468,-176.022,7.327,148.224
C06232=1223.384,344.785,-72.501,-176.020,7.329,148.224
C06233=1223.380,345.032,-72.532,-176.019,7.331,148.224
C06234=1223.375,345.280,-72.565,-176.017,7.335,148.225
C06235=1223.371,345.528,-72.596,-176.015,7.337,148.225
C06236=1223.367,345.776,-72.628,-176.013,7.340,148.225
C06237=1223.363,346.024,-72.660,-176.011,7.343,148.225
C06238=1223.359,346.271,-72.692,-176.009,7.346,148.225
C06239=1223.355,346.519,-72.724,-176.008,7.348,148.226
C06240=1223.351,346.768,-72.756,-176.006,7.352,148.226
C06241=1223.346,347.015,-72.788,-176.004,7.354,148.226
C06242=1223.342,347.263,-72.820,-176.002,7.357,148.226
C06243=1223.338,347.511,-72.852,-176.000,7.360,148.226
C06244=1223.334,347.759,-72.883,-175.998,7.362,148.226
C06245=1223.329,348.007,-72.916,-175.996,7.365,148.227
C06246=1223.326,348.255,-72.948,-175.994,7.368,148.227
C06247=1223.321,348.503,-72.981,-175.993,7.371,148.227
C06248=1223.317,348.750,-73.012,-175.991,7.373,148.227
C06249=1223.313,348.999,-73.045,-175.989,7.377,148.227
C06250=1223.309,349.247,-73.077,-175.987,7.379,148.228
C06251=1223.304,349.494,-73.109,-175.986,7.382,148.228
C06252=1223.300,349.742,-73.140,-175.984,7.384,148.228
C06253=1223.296,349.991,-73.173,-175.982,7.388,148.228
C06254=1223.292,350.238,-73.205,-175.980,7.390,148.228
C06255=1223.287,350.486,-73.238,-175.978,7.393,148.228
C06256=1223.284,350.734,-73.269,-175.977,7.396,148.229
C06257=1223.279,350.982,-73.302,-175.975,7.399,148.229
C06258=1223.275,351.229,-73.333,-175.973,7.401,148.229
C06259=1223.271,351.477,-73.366,-175.971,7.405,148.230
C06260=1223.267,351.725,-73.398,-175.970,7.407,148.230
C06261=1223.263,351.974,-73.431,-175.968,7.410,148.230
C06262=1223.258,352.221,-73.462,-175.966,7.412,148.230
C06263=1223.254,352.469,-73.495,-175.964,7.416,148.230
C06264=1223.250,352.717,-73.527,-175.963,7.418,148.231
C06265=1223.246,352.965,-73.560,-175.961,7.421,148.231
C06266=1223.243,353.212,-73.592,-175.959,7.424,148.231
C06267=1223.238,353.460,-73.624,-175.958,7.427,148.231
C06268=1223.233,353.708,-73.657,-175.956,7.429,148.231
C06269=1223.230,353.956,-73.689,-175.954,7.432,148.232
C06270=1223.225,354.204,-73.722,-175.952,7.435,148.232
C06271=1223.221,354.452,-73.753,-175.950,7.438,148.232
C06272=1223.217,354.699,-73.786,-175.949,7.440,148.232
C06273=1223.212,354.948,-73.819,-175.948,7.443,148.233
C06274=1223.209,355.196,-73.851,-175.945,7.446,148.233
C06275=1223.205,355.443,-73.884,-175.944,7.449,148.233
C06276=1223.201,355.691,-73.916,-175.942,7.452,148.233
C06277=1223.196,355.938,-73.948,-175.940,7.455,148.234
C06278=1223.192,356.187,-73.981,-175.939,7.458,148.234
C06279=1223.188,356.435,-74.013,-175.937,7.460,148.234
C06280=1223.184,356.683,-74.046,-175.936,7.463,148.234
C06281=1223.179,356.931,-74.078,-175.933,7.466,148.235
C06282=1223.175,357.178,-74.111,-175.932,7.469,148.235
C06283=1223.171,357.426,-74.143,-175.931,7.471,148.235
C06284=1223.167,357.674,-74.176,-175.929,7.474,148.235
C06285=1223.163,357.922,-74.208,-175.927,7.477,148.236
C06286=1223.159,358.169,-74.241,-175.926,7.480,148.236
C06287=1223.155,358.418,-74.274,-175.924,7.483,148.236
C06288=1223.151,358.665,-74.306,-175.922,7.485,148.236
C06289=1223.146,358.913,-74.338,-175.921,7.488,148.236
C06290=1223.142,359.161,-74.371,-175.919,7.491,148.237
C06291=1223.138,359.408,-74.404,-175.917,7.494,148.237
C06292=1223.134,359.656,-74.436,-175.916,7.496,148.237
C06293=1223.130,359.904,-74.469,-175.915,7.499,148.238
C06294=1223.126,360.152,-74.502,-175.912,7.503,148.238
C06295=1223.121,360.400,-74.535,-175.911,7.505,148.238
C06296=1223.118,360.648,-74.567,-175.910,7.508,148.238
C06297=1223.114,360.896,-74.600,-175.908,7.511,148.239
C06298=1223.109,361.143,-74.633,-175.907,7.513,148.239
C06299=1223.104,361.391,-74.665,-175.905,7.517,148.239
C06300=1223.101,361.639,-74.698,-175.903,7.519,148.239
C06301=1223.097,361.886,-74.731,-175.902,7.522,148.240
C06302=1223.092,362.135,-74.763,-175.900,7.525,148.240
C06303=1223.088,362.383,-74.797,-175.899,7.527,148.240
C06304=1223.084,362.630,-74.830,-175.897,7.531,148.241
C06305=1223.080,362.878,-74.862,-175.896,7.534,148.241
C06306=1223.076,363.126,-74.895,-175.894,7.536,148.241
C06307=1223.072,363.374,-74.928,-175.892,7.539,148.241
C06308=1223.068,363.622,-74.961,-175.891,7.541,148.242
C06309=1223.064,363.870,-74.994,-175.890,7.544,148.242
C06310=1223.059,364.118,-75.027,-175.888,7.548,148.242
C06311=1223.056,364.365,-75.059,-175.886,7.550,148.243
C06312=1223.051,364.612,-75.092,-175.885,7.553,148.243
C06313=1223.047,364.860,-75.124,-175.883,7.555,148.243
C06314=1223.043,365.108,-75.158,-175.882,7.558,148.244
C06315=1223.039,365.356,-75.191,-175.881,7.561,148.244
C06316=1223.034,365.604,-75.224,-175.879,7.565,148.244
C06317=1223.030,365.851,-75.257,-175.878,7.567,148.245
C06318=1223.027,366.099,-75.289,-175.876,7.570,148.245
C06319=1223.022,366.347,-75.322,-175.875,7.573,148.245
C06320=1223.018,366.595,-75.355,-175.873,7.575,148.245
C06321=1223.014,366.874,-75.393,-175.871,7.579,148.246
C06322=1223.009,367.155,-75.430,-175.870,7.582,148.246
C06323=1223.004,367.434,-75.467,-175.868,7.585,148.247
C06324=1223.000,367.714,-75.505,-175.867,7.588,148.247
C06325=1222.995,367.961,-75.538,-175.866,7.591,148.247
C06326=1222.991,368.209,-75.571,-175.864,7.593,148.248
C06327=1222.987,368.457,-75.604,-175.863,7.596,148.248
C06328=1222.983,368.705,-75.637,-175.862,7.599,148.248
C06329=1222.979,368.953,-75.670,-175.860,7.602,148.249
C06330=1222.974,369.201,-75.703,-175.858,7.605,148.249
C06331=1222.970,369.448,-75.736,-175.857,7.608,148.249
C06332=1222.966,369.696,-75.769,-175.856,7.610,148.250
C06333=1222.962,369.944,-75.802,-175.854,7.613,148.250
C06334=1222.958,370.192,-75.836,-175.853,7.616,148.250
C06335=1222.954,370.439,-75.869,-175.852,7.619,148.251
C06336=1222.950,370.687,-75.902,-175.850,7.621,148.251
C06337=1222.945,370.935,-75.935,-175.849,7.624,148.251
C06338=1222.942,371.183,-75.969,-175.848,7.627,148.252
C06339=1222.938,371.431,-76.002,-175.846,7.630,148.252
C06340=1222.934,371.679,-76.035,-175.845,7.632,148.252
C06341=1222.930,371.926,-76.068,-175.844,7.635,148.253
C06342=1222.925,372.174,-76.101,-175.843,7.638,148.253
C06343=1222.921,372.422,-76.134,-175.841,7.641,148.253
C06344=1222.917,372.670,-76.167,-175.840,7.643,148.254
C06345=1222.913,372.917,-76.201,-175.839,7.646,148.254
C06346=1222.909,373.165,-76.234,-175.838,7.649,148.254
C06347=1222.905,373.412,-76.268,-175.837,7.652,148.255
C06348=1222.901,373.660,-76.301,-175.835,7.654,148.255
C06349=1222.897,373.908,-76.334,-175.834,7.657,148.255
C06350=1222.893,374.155,-76.367,-175.833,7.660,148.256
C06351=1222.888,374.403,-76.401,-175.831,7.663,148.256
C06352=1222.884,374.651,-76.434,-175.830,7.666,148.257
C06353=1222.880,374.900,-76.468,-175.829,7.668,148.257
C06354=1222.876,375.147,-76.501,-175.828,7.671,148.257
C06355=1222.872,375.394,-76.535,-175.826,7.674,148.258
C06356=1222.868,375.642,-76.568,-175.825,7.677,148.258
C06357=1222.864,375.890,-76.601,-175.824,7.679,148.258
C06358=1222.860,376.138,-76.634,-175.823,7.682,148.259
C06359=1222.856,376.385,-76.668,-175.822,7.685,148.259
C06360=1222.851,376.633,-76.702,-175.821,7.687,148.260
C06361=1222.847,376.881,-76.735,-175.820,7.690,148.260
C06362=1222.843,377.129,-76.768,-175.819,7.693,148.260
C06363=1222.839,377.377,-76.801,-175.817,7.696,148.261
C06364=1222.835,377.624,-76.835,-175.816,7.698,148.261
C06365=1222.831,377.872,-76.868,-175.815,7.701,148.262
C06366=1222.826,378.120,-76.902,-175.814,7.704,148.262
C06367=1222.822,378.367,-76.935,-175.813,7.707,148.262
C06368=1222.818,378.614,-76.969,-175.812,7.710,148.263
C06369=1222.814,378.862,-77.002,-175.811,7.712,148.263
C06370=1222.811,379.111,-77.036,-175.810,7.714,148.263
C06371=1222.807,379.358,-77.070,-175.809,7.717,148.264
C06372=1222.802,379.606,-77.104,-175.807,7.720,148.264
C06373=1222.798,379.853,-77.137,-175.806,7.723,148.265
C06374=1222.794,380.101,-77.171,-175.805,7.726,148.265
C06375=1222.790,380.348,-77.204,-175.804,7.729,148.265
C06376=1222.786,380.597,-77.238,-175.803,7.730,148.266
C06377=1222.782,380.844,-77.272,-175.802,7.733,148.266
C06378=1222.778,381.092,-77.305,-175.801,7.736,148.267
C06379=1222.773,381.340,-77.338,-175.800,7.739,148.267
C06380=1222.769,381.587,-77.373,-175.798,7.742,148.267
C06381=1222.765,381.835,-77.406,-175.798,7.744,148.268
C06382=1222.761,382.083,-77.440,-175.797,7.747,148.268
C06383=1222.757,382.330,-77.473,-175.795,7.749,148.268
C06384=1222.752,382.578,-77.507,-175.794,7.752,148.269
C06385=1222.749,382.825,-77.541,-175.793,7.755,148.269
C06386=1222.745,383.073,-77.574,-175.792,7.757,148.270
C06387=1222.741,383.320,-77.608,-175.792,7.760,148.270
C06388=1222.736,383.569,-77.642,-175.791,7.763,148.271
C06389=1222.733,383.816,-77.676,-175.789,7.766,148.271
C06390=1222.728,384.064,-77.709,-175.789,7.768,148.271
C06391=1222.724,384.312,-77.743,-175.788,7.771,148.272
C06392=1222.720,384.559,-77.776,-175.786,7.773,148.272
C06393=1222.716,384.807,-77.810,-175.785,7.776,148.273
C06394=1222.712,385.055,-77.844,-175.785,7.778,148.273
C06395=1222.707,385.303,-77.878,-175.784,7.781,148.273
C06396=1222.704,385.550,-77.911,-175.783,7.784,148.274
C06397=1222.699,385.798,-77.946,-175.782,7.786,148.274
C06398=1222.696,386.046,-77.979,-175.781,7.789,148.275
C06399=1222.691,386.293,-78.013,-175.780,7.792,148.275
C06400=1222.687,386.541,-78.047,-175.779,7.795,148.275
C06401=1222.684,386.788,-78.081,-175.778,7.797,148.276
C06402=1222.679,387.036,-78.115,-175.777,7.800,148.276
C06403=1222.675,387.284,-78.149,-175.776,7.802,148.277
C06404=1222.671,387.531,-78.182,-175.775,7.804,148.277
C06405=1222.667,387.778,-78.216,-175.774,7.807,148.277
C06406=1222.663,388.027,-78.250,-175.773,7.810,148.278
C06407=1222.659,388.274,-78.284,-175.773,7.812,148.278
C06408=1222.654,388.522,-78.318,-175.772,7.815,148.279
C06409=1222.650,388.769,-78.352,-175.770,7.818,148.279
C06410=1222.647,389.017,-78.386,-175.770,7.820,148.280
C06411=1222.642,389.265,-78.420,-175.769,7.823,148.280
C06412=1222.638,389.512,-78.453,-175.768,7.825,148.281
C06413=1222.635,389.760,-78.488,-175.767,7.828,148.281
C06414=1222.630,390.008,-78.521,-175.766,7.831,148.281
C06415=1222.626,390.255,-78.555,-175.766,7.833,148.282
C06416=1222.622,390.503,-78.590,-175.765,7.836,148.282
C06417=1222.618,390.751,-78.623,-175.764,7.838,148.283
C06418=1222.614,390.999,-78.658,-175.763,7.841,148.283
C06419=1222.610,391.246,-78.692,-175.762,7.844,148.284
C06420=1222.606,391.494,-78.725,-175.762,7.846,148.284
C06421=1222.602,391.742,-78.760,-175.760,7.848,148.284
C06422=1222.598,391.989,-78.794,-175.760,7.851,148.285
C06423=1222.593,392.237,-78.827,-175.759,7.854,148.285
C06424=1222.590,392.485,-78.861,-175.758,7.856,148.286
C06425=1222.585,392.766,-78.901,-175.758,7.859,148.286
C06426=1222.580,393.048,-78.939,-175.756,7.862,148.287
C06427=1222.576,393.329,-78.978,-175.756,7.865,148.287
C06428=1222.570,393.611,-79.016,-175.755,7.867,148.288
C06429=1222.567,393.859,-79.051,-175.754,7.869,148.288
C06430=1222.563,394.106,-79.085,-175.753,7.873,148.289
C06431=1222.559,394.353,-79.119,-175.753,7.875,148.289
C06432=1222.555,394.602,-79.153,-175.751,7.877,148.289
C06433=1222.551,394.849,-79.187,-175.751,7.880,148.290
C06434=1222.546,395.097,-79.221,-175.750,7.882,148.290
C06435=1222.543,395.344,-79.256,-175.749,7.884,148.291
C06436=1222.538,395.593,-79.289,-175.749,7.888,148.291
C06437=1222.534,395.840,-79.323,-175.748,7.889,148.292
C06438=1222.530,396.088,-79.358,-175.747,7.892,148.292
C06439=1222.526,396.335,-79.392,-175.747,7.895,148.292
C06440=1222.522,396.582,-79.426,-175.745,7.897,148.293
C06441=1222.518,396.830,-79.461,-175.745,7.899,148.293
C06442=1222.514,397.078,-79.494,-175.744,7.902,148.294
C06443=1222.509,397.326,-79.529,-175.743,7.904,148.294
C06444=1222.506,397.573,-79.563,-175.743,7.906,148.294
C06445=1222.501,397.821,-79.598,-175.742,7.910,148.295
C06446=1222.497,398.068,-79.631,-175.741,7.912,148.295
C06447=1222.494,398.316,-79.666,-175.741,7.915,148.296
C06448=1222.490,398.563,-79.700,-175.740,7.917,148.296
C06449=1222.486,398.811,-79.735,-175.739,7.919,148.297
C06450=1222.481,399.059,-79.769,-175.739,7.922,148.297
C06451=1222.477,399.306,-79.803,-175.738,7.924,148.298
C06452=1222.473,399.554,-79.837,-175.737,7.927,148.298
C06453=1222.469,399.802,-79.871,-175.737,7.929,148.299
C06454=1222.465,400.049,-79.906,-175.736,7.931,148.299
C06455=1222.461,400.297,-79.941,-175.735,7.934,148.300
C06456=1222.457,400.544,-79.974,-175.735,7.936,148.300
C06457=1222.452,400.792,-80.009,-175.734,7.939,148.300
C06458=1222.449,401.039,-80.043,-175.733,7.941,148.301
C06459=1222.444,401.287,-80.078,-175.733,7.943,148.301
C06460=1222.441,401.535,-80.112,-175.732,7.946,148.302
C06461=1222.437,401.782,-80.146,-175.731,7.948,148.302
C06462=1222.432,402.030,-80.181,-175.731,7.950,148.302
C06463=1222.429,402.277,-80.215,-175.730,7.953,148.303
C06464=1222.424,402.525,-80.249,-175.729,7.955,148.303
C06465=1222.420,402.773,-80.284,-175.729,7.957,148.304
C06466=1222.417,403.020,-80.318,-175.728,7.959,148.304
C06467=1222.412,403.267,-80.353,-175.727,7.962,148.305
C06468=1222.408,403.516,-80.387,-175.727,7.964,148.305
C06469=1222.404,403.763,-80.421,-175.726,7.966,148.306
C06470=1222.400,404.011,-80.456,-175.725,7.969,148.306
C06471=1222.396,404.258,-80.491,-175.725,7.971,148.306
C06472=1222.392,404.505,-80.525,-175.724,7.973,148.307
C06473=1222.388,404.753,-80.559,-175.724,7.977,148.307
C06474=1222.383,405.001,-80.594,-175.723,7.979,148.308
C06475=1222.380,405.249,-80.628,-175.722,7.981,148.308
C06476=1222.375,405.496,-80.663,-175.722,7.983,148.309
C06477=1222.371,405.744,-80.697,-175.721,7.986,148.309
C06478=1222.368,405.991,-80.731,-175.721,7.988,148.310
C06479=1222.363,406.239,-80.766,-175.720,7.990,148.310
C06480=1222.359,406.487,-80.801,-175.720,7.992,148.310
C06481=1222.355,406.734,-80.834,-175.719,7.995,148.311
C06482=1222.351,406.982,-80.869,-175.718,7.997,148.311
C06483=1222.347,407.229,-80.904,-175.718,7.999,148.312
C06484=1222.344,407.477,-80.939,-175.717,8.001,148.312
C06485=1222.339,407.724,-80.973,-175.717,8.003,148.312
C06486=1222.335,407.972,-81.008,-175.716,8.006,148.313
C06487=1222.331,408.220,-81.042,-175.715,8.008,148.313
C06488=1222.327,408.467,-81.076,-175.715,8.011,148.314
C06489=1222.323,408.715,-81.111,-175.715,8.012,148.314
C06490=1222.318,408.962,-81.146,-175.714,8.014,148.315
C06491=1222.315,409.209,-81.181,-175.713,8.018,148.315
C06492=1222.311,409.457,-81.215,-175.713,8.020,148.315
C06493=1222.307,409.705,-81.250,-175.712,8.022,148.316
C06494=1222.302,409.952,-81.284,-175.712,8.024,148.316
C06495=1222.299,410.200,-81.319,-175.711,8.026,148.317
C06496=1222.294,410.448,-81.353,-175.711,8.028,148.317
C06497=1222.291,410.695,-81.389,-175.710,8.031,148.318
C06498=1222.286,410.943,-81.423,-175.710,8.033,148.318
C06499=1222.283,411.190,-81.457,-175.709,8.035,148.319
C06500=1222.278,411.438,-81.492,-175.709,8.037,148.319
C06501=1222.274,411.686,-81.527,-175.708,8.039,148.319
C06502=1222.270,411.933,-81.562,-175.707,8.041,148.320
C06503=1222.267,412.181,-81.596,-175.707,8.044,148.320
C06504=1222.262,412.428,-81.630,-175.706,8.046,148.321
C06505=1222.258,412.675,-81.665,-175.706,8.049,148.321
C06506=1222.254,412.924,-81.700,-175.705,8.051,148.322
C06507=1222.250,413.170,-81.735,-175.705,8.053,148.322
C06508=1222.246,413.418,-81.769,-175.704,8.055,148.322
C06509=1222.242,413.666,-81.804,-175.704,8.057,148.323
C06510=1222.238,413.913,-81.839,-175.703,8.059,148.323
C06511=1222.234,414.160,-81.874,-175.703,8.061,148.324
C06512=1222.230,414.409,-81.908,-175.702,8.063,148.324
C06513=1222.226,414.656,-81.942,-175.701,8.066,148.325
C06514=1222.222,414.903,-81.978,-175.701,8.068,148.325
C06515=1222.218,415.151,-82.012,-175.700,8.070,148.325
C06516=1222.214,415.399,-82.047,-175.700,8.072,148.326
C06517=1222.210,415.610,-82.077,-175.699,8.074,148.326
C06518=1222.207,415.822,-82.107,-175.699,8.076,148.326
C06519=1222.203,416.033,-82.137,-175.699,8.078,148.327
C06520=1222.200,416.245,-82.166,-175.698,8.080,148.327
C06521=1222.197,416.456,-82.196,-175.698,8.082,148.328
C06522=1222.193,416.668,-82.225,-175.698,8.083,148.328
C06523=1222.190,416.880,-82.255,-175.697,8.085,148.328
C06524=1222.190,417.091,-82.285,-175.696,8.087,148.329
C06525=1221.768,417.090,-82.319,-175.700,8.097,148.332
C06526=1221.768,416.878,-82.290,-175.700,8.096,148.332
C06527=1221.771,416.665,-82.259,-175.701,8.093,148.331
C06528=1221.774,416.453,-82.230,-175.701,8.092,148.331
C06529=1221.778,416.239,-82.200,-175.701,8.090,148.331
C06530=1221.781,416.027,-82.170,-175.702,8.088,148.331
C06531=1221.785,415.813,-82.140,-175.703,8.086,148.330
C06532=1221.789,415.601,-82.109,-175.703,8.085,148.330
C06533=1221.792,415.389,-82.080,-175.703,8.083,148.329
C06534=1221.796,415.140,-82.045,-175.704,8.081,148.329
C06535=1221.800,414.893,-82.011,-175.704,8.079,148.329
C06536=1221.804,414.645,-81.975,-175.704,8.077,148.328
C06537=1221.808,414.398,-81.941,-175.706,8.074,148.328
C06538=1221.812,414.150,-81.906,-175.706,8.071,148.327
C06539=1221.816,413.903,-81.872,-175.707,8.069,148.327
C06540=1221.820,413.655,-81.836,-175.707,8.068,148.327
C06541=1221.825,413.408,-81.802,-175.707,8.065,148.326
C06542=1221.828,413.160,-81.768,-175.708,8.063,148.326
C06543=1221.832,412.913,-81.733,-175.708,8.061,148.325
C06544=1221.836,412.665,-81.698,-175.709,8.059,148.325
C06545=1221.841,412.418,-81.663,-175.709,8.057,148.324
C06546=1221.845,412.170,-81.628,-175.710,8.054,148.324
C06547=1221.848,411.923,-81.594,-175.711,8.052,148.324
C06548=1221.852,411.675,-81.559,-175.711,8.050,148.323
C06549=1221.857,411.428,-81.524,-175.712,8.048,148.323
C06550=1221.861,411.179,-81.490,-175.712,8.046,148.322
C06551=1221.864,410.932,-81.456,-175.713,8.043,148.322
C06552=1221.868,410.684,-81.421,-175.713,8.041,148.321
C06553=1221.873,410.437,-81.386,-175.714,8.038,148.321
C06554=1221.877,410.189,-81.351,-175.715,8.036,148.320
C06555=1221.880,409.942,-81.317,-175.715,8.034,148.320
C06556=1221.884,409.694,-81.282,-175.715,8.032,148.320
C06557=1221.889,409.447,-81.248,-175.716,8.030,148.319
C06558=1221.893,409.199,-81.213,-175.716,8.028,148.319
C06559=1221.897,408.952,-81.178,-175.717,8.025,148.318
C06560=1221.900,408.704,-81.143,-175.718,8.023,148.318
C06561=1221.905,408.457,-81.109,-175.718,8.021,148.317
C06562=1221.910,408.209,-81.074,-175.719,8.019,148.317
C06563=1221.913,407.961,-81.040,-175.719,8.017,148.317
C06564=1221.917,407.714,-81.006,-175.720,8.014,148.316
C06565=1221.921,407.466,-80.971,-175.720,8.012,148.316
C06566=1221.925,407.219,-80.936,-175.721,8.010,148.315
C06567=1221.929,406.971,-80.902,-175.721,8.007,148.315
C06568=1221.933,406.724,-80.867,-175.722,8.005,148.314
C06569=1221.937,406.476,-80.832,-175.723,8.002,148.314
C06570=1221.941,406.229,-80.798,-175.723,8.000,148.313
C06571=1221.946,405.981,-80.764,-175.724,7.998,148.313
C06572=1221.950,405.733,-80.729,-175.724,7.996,148.313
C06573=1221.954,405.486,-80.695,-175.725,7.993,148.312
C06574=1221.958,405.238,-80.660,-175.726,7.991,148.312
C06575=1221.962,404.990,-80.626,-175.726,7.989,148.311
C06576=1221.965,404.743,-80.592,-175.727,7.987,148.311
C06577=1221.970,404.496,-80.556,-175.727,7.984,148.310
C06578=1221.974,404.248,-80.522,-175.728,7.982,148.310
C06579=1221.977,404.000,-80.488,-175.729,7.980,148.310
C06580=1221.982,403.753,-80.453,-175.729,7.977,148.309
C06581=1221.986,403.505,-80.418,-175.730,7.975,148.309
C06582=1221.990,403.258,-80.385,-175.730,7.972,148.308
C06583=1221.994,403.010,-80.350,-175.731,7.971,148.308
C06584=1221.998,402.762,-80.315,-175.732,7.968,148.307
C06585=1222.002,402.515,-80.281,-175.732,7.965,148.307
C06586=1222.006,402.267,-80.247,-175.733,7.963,148.307
C06587=1222.011,402.020,-80.212,-175.734,7.960,148.306
C06588=1222.014,401.772,-80.178,-175.734,7.958,148.306
C06589=1222.019,401.524,-80.143,-175.735,7.956,148.305
C06590=1222.022,401.277,-80.110,-175.736,7.953,148.305
C06591=1222.026,401.029,-80.075,-175.736,7.951,148.304
C06592=1222.031,400.782,-80.040,-175.737,7.949,148.304
C06593=1222.035,400.534,-80.007,-175.738,7.946,148.303
C06594=1222.039,400.286,-79.972,-175.738,7.944,148.303
C06595=1222.043,400.039,-79.938,-175.739,7.941,148.303
C06596=1222.047,399.791,-79.904,-175.740,7.939,148.302
C06597=1222.051,399.543,-79.869,-175.740,7.937,148.302
C06598=1222.055,399.296,-79.835,-175.741,7.934,148.301
C06599=1222.059,399.048,-79.800,-175.742,7.932,148.301
C06600=1222.063,398.801,-79.767,-175.742,7.930,148.300
C06601=1222.068,398.554,-79.732,-175.743,7.927,148.300
C06602=1222.072,398.305,-79.697,-175.744,7.925,148.300
C06603=1222.075,398.058,-79.663,-175.744,7.922,148.299
C06604=1222.079,397.810,-79.629,-175.745,7.920,148.299
C06605=1222.083,397.562,-79.595,-175.746,7.917,148.298
C06606=1222.088,397.315,-79.561,-175.746,7.915,148.298
C06607=1222.091,397.067,-79.527,-175.747,7.913,148.297
C06608=1222.096,396.820,-79.492,-175.748,7.910,148.297
C06609=1222.100,396.573,-79.458,-175.748,7.908,148.296
C06610=1222.104,396.325,-79.423,-175.750,7.905,148.296
C06611=1222.109,396.077,-79.390,-175.750,7.903,148.296
C06612=1222.112,395.829,-79.356,-175.751,7.900,148.295
C06613=1222.116,395.581,-79.321,-175.752,7.898,148.295
C06614=1222.120,395.334,-79.287,-175.752,7.895,148.294
C06615=1222.125,395.087,-79.253,-175.753,7.893,148.294
C06616=1222.128,394.839,-79.218,-175.754,7.890,148.293
C06617=1222.133,394.591,-79.185,-175.754,7.888,148.293
C06618=1222.137,394.344,-79.151,-175.756,7.885,148.292
C06619=1222.141,394.096,-79.116,-175.756,7.883,148.292
C06620=1222.144,393.849,-79.082,-175.757,7.880,148.292
C06621=1222.149,393.601,-79.048,-175.758,7.878,148.291
C06622=1222.153,393.319,-79.010,-175.758,7.875,148.291
C06623=1222.158,393.038,-78.970,-175.760,7.872,148.290
C06624=1222.163,392.756,-78.932,-175.760,7.869,148.290
C06625=1222.167,392.474,-78.893,-175.761,7.866,148.289
C06626=1222.172,392.226,-78.859,-175.762,7.864,148.289
C06627=1222.175,391.978,-78.825,-175.763,7.861,148.288
C06628=1222.180,391.731,-78.791,-175.763,7.859,148.288
C06629=1222.184,391.483,-78.757,-175.765,7.856,148.288
C06630=1222.188,391.235,-78.723,-175.765,7.854,148.287
C06631=1222.192,390.988,-78.689,-175.766,7.851,148.287
C06632=1222.195,390.741,-78.655,-175.767,7.848,148.286
C06633=1222.200,390.493,-78.621,-175.768,7.846,148.286
C06634=1222.204,390.245,-78.587,-175.769,7.843,148.285
C06635=1222.208,389.998,-78.552,-175.769,7.841,148.285
C06636=1222.212,389.750,-78.519,-175.770,7.838,148.284
C06637=1222.216,389.502,-78.484,-175.772,7.835,148.284
C06638=1222.220,389.254,-78.451,-175.772,7.833,148.284
C06639=1222.224,389.007,-78.417,-175.773,7.830,148.283
C06640=1222.229,388.760,-78.383,-175.774,7.828,148.283
C06641=1222.232,388.511,-78.349,-175.775,7.826,148.282
C06642=1222.237,388.264,-78.315,-175.775,7.822,148.282
C06643=1222.241,388.017,-78.281,-175.776,7.820,148.281
C06644=1222.245,387.769,-78.248,-175.777,7.818,148.281
C06645=1222.249,387.521,-78.213,-175.778,7.815,148.281
C06646=1222.253,387.273,-78.180,-175.779,7.813,148.280
C06647=1222.257,387.026,-78.146,-175.780,7.810,148.280
C06648=1222.262,386.778,-78.112,-175.781,7.807,148.279
C06649=1222.265,386.530,-78.078,-175.782,7.805,148.279
C06650=1222.269,386.283,-78.044,-175.783,7.802,148.279
C06651=1222.274,386.035,-78.010,-175.784,7.799,148.278
C06652=1222.277,385.788,-77.977,-175.785,7.796,148.278
C06653=1222.282,385.540,-77.943,-175.785,7.794,148.277
C06654=1222.286,385.292,-77.909,-175.786,7.791,148.277
C06655=1222.290,385.044,-77.875,-175.788,7.789,148.276
C06656=1222.294,384.797,-77.841,-175.788,7.787,148.276
C06657=1222.298,384.549,-77.808,-175.789,7.784,148.276
C06658=1222.302,384.301,-77.774,-175.790,7.781,148.275
C06659=1222.306,384.053,-77.740,-175.791,7.778,148.275
C06660=1222.310,383.806,-77.706,-175.792,7.776,148.274
C06661=1222.314,383.558,-77.673,-175.793,7.773,148.274
C06662=1222.319,383.311,-77.640,-175.794,7.770,148.274
C06663=1222.323,383.063,-77.605,-175.796,7.767,148.273
C06664=1222.327,382.815,-77.572,-175.796,7.765,148.273
C06665=1222.330,382.568,-77.538,-175.797,7.763,148.272
C06666=1222.335,382.320,-77.504,-175.799,7.760,148.272
C06667=1222.339,382.073,-77.470,-175.799,7.757,148.271
C06668=1222.343,381.824,-77.437,-175.800,7.754,148.271
C06669=1222.347,381.576,-77.403,-175.801,7.752,148.271
C06670=1222.351,381.329,-77.369,-175.802,7.749,148.270
C06671=1222.356,381.081,-77.336,-175.803,7.746,148.270
C06672=1222.359,380.834,-77.302,-175.805,7.743,148.270
C06673=1222.364,380.586,-77.269,-175.806,7.741,148.269
C06674=1222.368,380.338,-77.235,-175.807,7.738,148.269
C06675=1222.372,380.091,-77.201,-175.808,7.736,148.268
C06676=1222.376,379.843,-77.168,-175.809,7.733,148.268
C06677=1222.380,379.595,-77.135,-175.810,7.730,148.268
C06678=1222.384,379.348,-77.101,-175.811,7.727,148.267
C06679=1222.389,379.100,-77.067,-175.812,7.724,148.267
C06680=1222.392,378.852,-77.033,-175.814,7.722,148.266
C06681=1222.396,378.604,-77.000,-175.815,7.719,148.266
C06682=1222.400,378.357,-76.966,-175.815,7.717,148.266
C06683=1222.404,378.109,-76.933,-175.817,7.714,148.265
C06684=1222.409,377.861,-76.899,-175.818,7.711,148.265
C06685=1222.413,377.614,-76.866,-175.819,7.708,148.265
C06686=1222.417,377.366,-76.832,-175.820,7.706,148.264
C06687=1222.421,377.118,-76.799,-175.821,7.703,148.264
C06688=1222.425,376.870,-76.766,-175.822,7.700,148.263
C06689=1222.429,376.623,-76.732,-175.824,7.697,148.263
C06690=1222.434,376.375,-76.698,-175.825,7.694,148.263
C06691=1222.438,376.127,-76.665,-175.826,7.691,148.262
C06692=1222.442,375.879,-76.632,-175.827,7.689,148.262
C06693=1222.446,375.632,-76.599,-175.828,7.687,148.262
C06694=1222.450,375.384,-76.565,-175.829,7.684,148.261
C06695=1222.454,375.137,-76.532,-175.831,7.681,148.261
C06696=1222.458,374.889,-76.498,-175.832,7.679,148.260
C06697=1222.462,374.641,-76.465,-175.833,7.676,148.260
C06698=1222.466,374.393,-76.431,-175.834,7.673,148.260
C06699=1222.471,374.145,-76.398,-175.835,7.670,148.259
C06700=1222.474,373.898,-76.364,-175.836,7.667,148.259
C06701=1222.479,373.650,-76.331,-175.838,7.665,148.259
C06702=1222.483,373.402,-76.298,-175.839,7.662,148.258
C06703=1222.487,373.155,-76.265,-175.840,7.659,148.258
C06704=1222.491,372.907,-76.232,-175.842,7.656,148.257
C06705=1222.495,372.659,-76.198,-175.843,7.653,148.257
C06706=1222.499,372.411,-76.165,-175.844,7.651,148.257
C06707=1222.503,372.164,-76.132,-175.846,7.648,148.256
C06708=1222.508,371.916,-76.099,-175.847,7.645,148.256
C06709=1222.512,371.668,-76.066,-175.848,7.642,148.256
C06710=1222.515,371.420,-76.032,-175.849,7.640,148.255
C06711=1222.519,371.172,-75.999,-175.851,7.637,148.255
C06712=1222.523,370.924,-75.966,-175.852,7.634,148.255
C06713=1222.528,370.677,-75.933,-175.853,7.631,148.254
C06714=1222.532,370.429,-75.900,-175.854,7.629,148.254
C06715=1222.536,370.181,-75.866,-175.856,7.626,148.254
C06716=1222.540,369.933,-75.833,-175.857,7.623,148.253
C06717=1222.544,369.686,-75.800,-175.859,7.620,148.253
C06718=1222.548,369.438,-75.767,-175.860,7.617,148.253
C06719=1222.552,369.190,-75.734,-175.862,7.614,148.252
C06720=1222.557,368.942,-75.701,-175.863,7.611,148.252
C06721=1222.561,368.695,-75.668,-175.864,7.609,148.252
C06722=1222.565,368.447,-75.634,-175.866,7.606,148.251
C06723=1222.569,368.199,-75.601,-175.867,7.603,148.251
C06724=1222.573,367.952,-75.568,-175.868,7.601,148.251
C06725=1222.577,367.704,-75.535,-175.870,7.598,148.250
C06726=1222.582,367.424,-75.497,-175.871,7.594,148.250
C06727=1222.587,367.144,-75.461,-175.873,7.592,148.250
C06728=1222.591,366.864,-75.423,-175.875,7.588,148.249
C06729=1222.596,366.585,-75.386,-175.876,7.585,148.249
C06730=1222.600,366.336,-75.353,-175.878,7.583,148.249
C06731=1222.605,366.089,-75.320,-175.879,7.579,148.248
C06732=1222.609,365.841,-75.287,-175.881,7.577,148.248
C06733=1222.613,365.593,-75.254,-175.882,7.574,148.248
C06734=1222.617,365.346,-75.220,-175.883,7.571,148.247
C06735=1222.620,365.098,-75.188,-175.885,7.568,148.247
C06736=1222.625,364.850,-75.155,-175.886,7.566,148.247
C06737=1222.629,364.602,-75.122,-175.888,7.563,148.246
C06738=1222.633,364.354,-75.089,-175.889,7.559,148.246
C06739=1222.637,364.107,-75.056,-175.891,7.557,148.246
C06740=1222.641,363.859,-75.023,-175.892,7.554,148.245
C06741=1222.645,363.611,-74.991,-175.894,7.552,148.245
C06742=1222.649,363.363,-74.958,-175.895,7.549,148.245
C06743=1222.654,363.116,-74.925,-175.897,7.545,148.245
C06744=1222.658,362.868,-74.893,-175.898,7.543,148.244
C06745=1222.663,362.620,-74.859,-175.900,7.540,148.244
C06746=1222.667,362.372,-74.826,-175.902,7.537,148.244
C06747=1222.670,362.125,-74.794,-175.903,7.535,148.243
C06748=1222.675,361.876,-74.761,-175.904,7.532,148.243
C06749=1222.679,361.629,-74.728,-175.906,7.528,148.243
C06750=1222.683,361.381,-74.695,-175.908,7.526,148.243
C06751=1222.687,361.133,-74.663,-175.909,7.523,148.242
C06752=1222.691,360.885,-74.630,-175.911,7.521,148.242
C06753=1222.695,360.637,-74.598,-175.913,7.517,148.242
C06754=1222.699,360.389,-74.564,-175.914,7.514,148.241
C06755=1222.704,360.142,-74.532,-175.916,7.512,148.241
C06756=1222.708,359.894,-74.500,-175.917,7.509,148.241
C06757=1222.712,359.646,-74.467,-175.918,7.507,148.241
C06758=1222.716,359.398,-74.434,-175.921,7.503,148.240
C06759=1222.720,359.150,-74.401,-175.922,7.501,148.240
C06760=1222.724,358.903,-74.368,-175.923,7.498,148.240
C06761=1222.728,358.655,-74.336,-175.925,7.495,148.240
C06762=1222.732,358.407,-74.303,-175.927,7.492,148.239
C06763=1222.737,358.159,-74.271,-175.928,7.489,148.239
C06764=1222.741,357.912,-74.238,-175.930,7.487,148.239
C06765=1222.745,357.663,-74.206,-175.932,7.484,148.239
C06766=1222.749,357.416,-74.173,-175.934,7.481,148.238
C06767=1222.753,357.168,-74.141,-175.935,7.478,148.238
C06768=1222.757,356.920,-74.108,-175.937,7.475,148.238
C06769=1222.762,356.672,-74.075,-175.938,7.473,148.238
C06770=1222.766,356.425,-74.043,-175.940,7.469,148.237
C06771=1222.770,356.176,-74.011,-175.942,7.467,148.237
C06772=1222.774,355.928,-73.979,-175.943,7.464,148.237
C06773=1222.778,355.681,-73.946,-175.945,7.462,148.237
C06774=1222.782,355.432,-73.913,-175.947,7.458,148.236
C06775=1222.786,355.186,-73.881,-175.948,7.455,148.236
C06776=1222.791,354.937,-73.848,-175.950,7.453,148.236
C06777=1222.795,354.690,-73.815,-175.952,7.450,148.236
C06778=1222.799,354.442,-73.783,-175.954,7.447,148.235
C06779=1222.803,354.193,-73.751,-175.955,7.444,148.235
C06780=1222.807,353.946,-73.719,-175.957,7.442,148.235
C06781=1222.812,353.698,-73.686,-175.959,7.438,148.235
C06782=1222.816,353.450,-73.654,-175.960,7.436,148.234
C06783=1222.819,353.202,-73.621,-175.962,7.433,148.234
C06784=1222.824,352.954,-73.589,-175.964,7.431,148.234
C06785=1222.828,352.707,-73.557,-175.966,7.427,148.234
C06786=1222.833,352.458,-73.525,-175.967,7.425,148.234
C06787=1222.836,352.211,-73.492,-175.969,7.422,148.233
C06788=1222.840,351.963,-73.460,-175.971,7.419,148.233
C06789=1222.846,351.715,-73.428,-175.973,7.416,148.233
C06790=1222.849,351.467,-73.395,-175.974,7.414,148.233
C06791=1222.853,351.219,-73.363,-175.976,7.410,148.232
C06792=1222.857,350.971,-73.331,-175.978,7.408,148.232
C06793=1222.862,350.723,-73.299,-175.980,7.405,148.232
C06794=1222.866,350.475,-73.267,-175.981,7.403,148.232
C06795=1222.870,350.228,-73.234,-175.983,7.399,148.232
C06796=1222.874,349.980,-73.202,-175.985,7.397,148.231
C06797=1222.879,349.732,-73.170,-175.987,7.394,148.231
C06798=1222.882,349.484,-73.138,-175.989,7.391,148.231
C06799=1222.887,349.236,-73.106,-175.990,7.388,148.231
C06800=1222.891,348.988,-73.074,-175.992,7.386,148.231
C06801=1222.895,348.741,-73.042,-175.994,7.382,148.230
C06802=1222.899,348.492,-73.009,-175.996,7.380,148.230
C06803=1222.903,348.244,-72.977,-175.998,7.377,148.230
C06804=1222.908,347.997,-72.945,-176.000,7.374,148.230
C06805=1222.911,347.749,-72.914,-176.001,7.372,148.230
C06806=1222.916,347.500,-72.881,-176.003,7.369,148.230
C06807=1222.920,347.253,-72.850,-176.005,7.366,148.229
C06808=1222.925,347.005,-72.817,-176.007,7.363,148.229
C06809=1222.928,346.757,-72.785,-176.008,7.361,148.229
C06810=1222.933,346.509,-72.754,-176.010,7.358,148.229
C06811=1222.937,346.261,-72.721,-176.013,7.355,148.229
C06812=1222.941,346.013,-72.690,-176.014,7.353,148.229
C06813=1222.945,345.766,-72.658,-176.016,7.350,148.228
C06814=1222.950,345.517,-72.626,-176.018,7.347,148.228
C06815=1222.953,345.269,-72.594,-176.020,7.344,148.228
C06816=1222.958,345.022,-72.562,-176.021,7.342,148.228
C06817=1222.962,344.774,-72.530,-176.024,7.338,148.228
C06818=1222.966,344.526,-72.498,-176.025,7.336,148.227
C06819=1222.971,344.278,-72.466,-176.027,7.332,148.227
C06820=1222.975,344.030,-72.434,-176.030,7.330,148.227
C06821=1222.978,343.782,-72.402,-176.031,7.328,148.227
C06822=1222.983,343.534,-72.370,-176.033,7.324,148.227
C06823=1222.987,343.286,-72.338,-176.035,7.322,148.227
C06824=1222.991,343.039,-72.307,-176.037,7.319,148.226
C06825=1222.996,342.790,-72.275,-176.039,7.316,148.226
C06826=1223.000,342.542,-72.243,-176.041,7.314,148.226
C06827=1223.004,342.294,-72.212,-176.043,7.311,148.226
C06828=1223.008,342.046,-72.180,-176.045,7.308,148.226
C06829=1223.013,341.799,-72.148,-176.046,7.305,148.226
C06830=1223.017,341.521,-72.112,-176.049,7.302,148.225
C06831=1223.022,341.243,-72.077,-176.051,7.300,148.225
C06832=1223.027,340.965,-72.041,-176.053,7.296,148.225
C06833=1223.031,340.688,-72.006,-176.055,7.293,148.225
C06834=1223.035,340.439,-71.974,-176.057,7.290,148.225
C06835=1223.039,340.192,-71.943,-176.059,7.287,148.225
C06836=1223.044,339.943,-71.911,-176.061,7.285,148.225
C06837=1223.048,339.696,-71.879,-176.063,7.282,148.224
C06838=1223.052,339.447,-71.848,-176.065,7.279,148.224
C06839=1223.056,339.200,-71.816,-176.067,7.277,148.224
C06840=1223.060,338.952,-71.785,-176.069,7.273,148.224
C06841=1223.065,338.704,-71.754,-176.071,7.271,148.224
C06842=1223.069,338.456,-71.721,-176.073,7.269,148.224
C06843=1223.073,338.208,-71.690,-176.075,7.265,148.224
C06844=1223.078,337.960,-71.659,-176.077,7.263,148.223
C06845=1223.081,337.712,-71.627,-176.079,7.260,148.223
C06846=1223.086,337.464,-71.596,-176.081,7.257,148.223
C06847=1223.090,337.216,-71.564,-176.083,7.255,148.223
C06848=1223.094,336.968,-71.533,-176.085,7.252,148.223
C06849=1223.098,336.720,-71.500,-176.087,7.249,148.223
C06850=1223.103,336.472,-71.470,-176.088,7.246,148.223
C06851=1223.107,336.224,-71.438,-176.091,7.243,148.223
C06852=1223.111,335.976,-71.407,-176.093,7.241,148.223
C06853=1223.115,335.728,-71.375,-176.094,7.238,148.222
C06854=1223.120,335.480,-71.344,-176.097,7.235,148.222
C06855=1223.123,335.232,-71.313,-176.099,7.233,148.222
C06856=1223.128,334.984,-71.282,-176.100,7.230,148.222
C06857=1223.132,334.736,-71.250,-176.103,7.227,148.222
C06858=1223.136,334.489,-71.219,-176.105,7.225,148.222
C06859=1223.140,334.240,-71.187,-176.107,7.222,148.222
C06860=1223.145,333.992,-71.157,-176.109,7.219,148.222
C06861=1223.148,333.744,-71.125,-176.111,7.217,148.222
C06862=1223.154,333.496,-71.093,-176.113,7.213,148.221
C06863=1223.158,333.248,-71.062,-176.115,7.211,148.221
C06864=1223.162,333.000,-71.031,-176.117,7.209,148.221
C06865=1223.166,332.752,-70.999,-176.119,7.205,148.221
C06866=1223.170,332.504,-70.968,-176.121,7.203,148.221
C06867=1223.175,332.256,-70.937,-176.123,7.200,148.221
C06868=1223.179,332.008,-70.906,-176.125,7.198,148.221
C06869=1223.183,331.760,-70.875,-176.127,7.195,148.221
C06870=1223.187,331.513,-70.844,-176.130,7.192,148.221
C06871=1223.191,331.264,-70.813,-176.131,7.189,148.221
C06872=1223.195,331.016,-70.782,-176.133,7.187,148.221
C06873=1223.199,330.768,-70.750,-176.136,7.184,148.220
C06874=1223.204,330.520,-70.719,-176.138,7.182,148.220
C06875=1223.208,330.271,-70.688,-176.140,7.178,148.220
C06876=1223.212,330.024,-70.657,-176.142,7.176,148.220
C06877=1223.217,329.776,-70.626,-176.144,7.174,148.220
C06878=1223.221,329.527,-70.595,-176.146,7.170,148.220
C06879=1223.225,329.280,-70.563,-176.148,7.168,148.220
C06880=1223.230,329.032,-70.533,-176.151,7.165,148.220
C06881=1223.234,328.784,-70.502,-176.152,7.162,148.220
C06882=1223.238,328.536,-70.471,-176.154,7.160,148.220
C06883=1223.241,328.288,-70.440,-176.157,7.157,148.220
C06884=1223.246,328.040,-70.409,-176.159,7.155,148.220
C06885=1223.250,327.792,-70.378,-176.161,7.152,148.220
C06886=1223.254,327.543,-70.347,-176.163,7.149,148.219
C06887=1223.259,327.295,-70.316,-176.165,7.147,148.219
C06888=1223.263,327.048,-70.285,-176.167,7.143,148.219
C06889=1223.267,326.799,-70.254,-176.169,7.141,148.219
C06890=1223.271,326.552,-70.223,-176.171,7.139,148.219
C06891=1223.276,326.304,-70.193,-176.174,7.136,148.219
C06892=1223.280,326.055,-70.161,-176.176,7.133,148.219
C06893=1223.284,325.807,-70.131,-176.178,7.130,148.219
C06894=1223.289,325.559,-70.100,-176.180,7.128,148.219
C06895=1223.292,325.311,-70.069,-176.182,7.126,148.219
C06896=1223.297,325.063,-70.039,-176.184,7.122,148.219
C06897=1223.301,324.815,-70.007,-176.186,7.120,148.219
C06898=1223.305,324.567,-69.976,-176.188,7.117,148.219
C06899=1223.309,324.319,-69.946,-176.191,7.114,148.219
C06900=1223.314,324.071,-69.915,-176.193,7.112,148.219
C06901=1223.318,323.823,-69.884,-176.195,7.109,148.218
C06902=1223.322,323.575,-69.853,-176.197,7.107,148.218
C06903=1223.326,323.327,-69.823,-176.199,7.104,148.219
C06904=1223.331,323.079,-69.792,-176.201,7.101,148.218
C06905=1223.335,322.830,-69.761,-176.203,7.099,148.218
C06906=1223.340,322.582,-69.730,-176.206,7.096,148.218
C06907=1223.343,322.335,-69.700,-176.208,7.094,148.218
C06908=1223.347,322.086,-69.669,-176.210,7.091,148.218
C06909=1223.352,321.838,-69.638,-176.213,7.088,148.218
C06910=1223.356,321.590,-69.609,-176.215,7.086,148.218
C06911=1223.361,321.342,-69.578,-176.216,7.083,148.218
C06912=1223.365,321.093,-69.547,-176.219,7.080,148.218
C06913=1223.369,320.846,-69.517,-176.221,7.078,148.218
C06914=1223.373,320.598,-69.486,-176.224,7.075,148.218
C06915=1223.378,320.350,-69.455,-176.225,7.072,148.218
C06916=1223.382,320.102,-69.425,-176.227,7.070,148.218
C06917=1223.386,319.853,-69.394,-176.230,7.067,148.218
C06918=1223.390,319.605,-69.365,-176.232,7.065,148.218
C06919=1223.395,319.357,-69.334,-176.234,7.061,148.218
C06920=1223.399,319.109,-69.303,-176.236,7.059,148.218
C06921=1223.402,318.861,-69.272,-176.239,7.057,148.218
C06922=1223.407,318.613,-69.242,-176.241,7.054,148.218
C06923=1223.411,318.365,-69.212,-176.243,7.051,148.218
C06924=1223.416,318.117,-69.181,-176.245,7.049,148.218
C06925=1223.421,317.869,-69.151,-176.248,7.046,148.218
C06926=1223.424,317.620,-69.120,-176.250,7.044,148.218
C06927=1223.429,317.372,-69.090,-176.252,7.041,148.218
C06928=1223.433,317.124,-69.060,-176.254,7.038,148.218
C06929=1223.437,316.876,-69.029,-176.256,7.036,148.218
C06930=1223.441,316.628,-69.000,-176.259,7.033,148.218
C06931=1223.446,316.380,-68.969,-176.261,7.031,148.218
C06932=1223.449,316.132,-68.938,-176.264,7.028,148.218
C06933=1223.454,315.884,-68.908,-176.266,7.026,148.218
C06934=1223.458,315.608,-68.875,-176.268,7.022,148.218
C06935=1223.464,315.332,-68.841,-176.270,7.020,148.218
C06936=1223.469,315.056,-68.807,-176.273,7.017,148.218
C06937=1223.473,314.781,-68.774,-176.275,7.014,148.218
C06938=1223.478,314.532,-68.744,-176.277,7.012,148.218
C06939=1223.482,314.284,-68.713,-176.280,7.009,148.218
C06940=1223.486,314.036,-68.683,-176.282,7.006,148.218
C06941=1223.490,313.788,-68.653,-176.284,7.004,148.218
C06942=1223.494,313.539,-68.623,-176.287,7.001,148.218
C06943=1223.499,313.291,-68.593,-176.289,6.999,148.218
C06944=1223.503,313.043,-68.563,-176.291,6.996,148.218
C06945=1223.507,312.795,-68.532,-176.293,6.993,148.218
C06946=1223.511,312.547,-68.503,-176.295,6.991,148.218
C06947=1223.516,312.299,-68.472,-176.298,6.988,148.218
C06948=1223.520,312.050,-68.443,-176.300,6.986,148.218
C06949=1223.524,311.803,-68.412,-176.302,6.984,148.218
C06950=1223.529,311.554,-68.382,-176.305,6.981,148.218
C06951=1223.533,311.307,-68.352,-176.307,6.978,148.218
C06952=1223.537,311.058,-68.323,-176.310,6.975,148.218
C06953=1223.542,310.810,-68.292,-176.312,6.973,148.218
C06954=1223.546,310.562,-68.263,-176.314,6.971,148.218
C06955=1223.550,310.313,-68.231,-176.317,6.968,148.218
C06956=1223.554,310.065,-68.202,-176.318,6.965,148.218
C06957=1223.558,309.817,-68.173,-176.320,6.963,148.218
C06958=1223.563,309.569,-68.142,-176.323,6.960,148.218
C06959=1223.567,309.321,-68.112,-176.325,6.958,148.218
C06960=1223.571,309.072,-68.083,-176.327,6.956,148.218
C06961=1223.575,308.825,-68.053,-176.330,6.953,148.218
C06962=1223.580,308.576,-68.023,-176.332,6.950,148.218
C06963=1223.584,308.328,-67.993,-176.335,6.947,148.218
C06964=1223.588,308.080,-67.963,-176.337,6.945,148.218
C06965=1223.593,307.832,-67.933,-176.339,6.943,148.218
C06966=1223.597,307.583,-67.904,-176.342,6.940,148.218
C06967=1223.601,307.335,-67.874,-176.344,6.938,148.218
C06968=1223.605,307.088,-67.844,-176.346,6.935,148.218
C06969=1223.610,306.839,-67.814,-176.348,6.932,148.218
C06970=1223.614,306.591,-67.784,-176.351,6.930,148.218
C06971=1223.619,306.342,-67.755,-176.353,6.928,148.218
C06972=1223.622,306.095,-67.725,-176.355,6.925,148.218
C06973=1223.627,305.846,-67.695,-176.357,6.923,148.218
C06974=1223.632,305.598,-67.665,-176.360,6.920,148.219
C06975=1223.636,305.350,-67.636,-176.362,6.917,148.219
C06976=1223.641,305.102,-67.607,-176.364,6.915,148.219
C06977=1223.645,304.854,-67.577,-176.367,6.912,148.219
C06978=1223.650,304.605,-67.547,-176.370,6.910,148.219
C06979=1223.653,304.358,-67.517,-176.372,6.908,148.219
C06980=1223.658,304.109,-67.488,-176.374,6.905,148.219
C06981=1223.662,303.861,-67.458,-176.376,6.903,148.219
C06982=1223.666,303.613,-67.429,-176.379,6.901,148.219
C06983=1223.670,303.365,-67.399,-176.381,6.897,148.219
C06984=1223.674,303.116,-67.370,-176.383,6.895,148.219
C06985=1223.679,302.868,-67.340,-176.385,6.893,148.219
C06986=1223.683,302.619,-67.310,-176.388,6.890,148.219
C06987=1223.688,302.371,-67.281,-176.390,6.888,148.219
C06988=1223.692,302.123,-67.251,-176.392,6.886,148.219
C06989=1223.697,301.875,-67.222,-176.395,6.883,148.219
C06990=1223.701,301.627,-67.193,-176.397,6.880,148.219
C06991=1223.705,301.379,-67.163,-176.400,6.878,148.220
C06992=1223.709,301.130,-67.134,-176.402,6.875,148.220
C06993=1223.713,300.882,-67.105,-176.404,6.873,148.220
C06994=1223.718,300.634,-67.075,-176.407,6.871,148.220
C06995=1223.722,300.386,-67.046,-176.409,6.868,148.220
C06996=1223.726,300.137,-67.016,-176.411,6.866,148.220
C06997=1223.730,299.889,-66.987,-176.413,6.863,148.220
C06998=1223.735,299.642,-66.958,-176.416,6.860,148.220
C06999=1223.739,299.393,-66.928,-176.419,6.859,148.220
C07000=1223.743,299.145,-66.899,-176.421,6.856,148.220
C07001=1223.748,298.896,-66.870,-176.423,6.853,148.220
C07002=1223.752,298.648,-66.841,-176.426,6.851,148.220
C07003=1223.756,298.400,-66.811,-176.428,6.849,148.220
C07004=1223.761,298.152,-66.782,-176.430,6.846,148.220
C07005=1223.765,297.904,-66.753,-176.432,6.844,148.220
C07006=1223.769,297.656,-66.723,-176.435,6.842,148.221
C07007=1223.774,297.407,-66.694,-176.438,6.839,148.221
C07008=1223.778,297.158,-66.665,-176.440,6.836,148.221
C07009=1223.782,296.910,-66.635,-176.442,6.834,148.221
C07010=1223.787,296.663,-66.606,-176.445,6.831,148.221
C07011=1223.791,296.414,-66.578,-176.447,6.829,148.221
C07012=1223.796,296.165,-66.548,-176.449,6.827,148.221
C07013=1223.800,295.917,-66.519,-176.452,6.824,148.221
C07014=1223.804,295.669,-66.489,-176.454,6.822,148.221
C07015=1223.809,295.421,-66.461,-176.456,6.820,148.221
C07016=1223.813,295.172,-66.431,-176.459,6.817,148.222
C07017=1223.817,294.924,-66.403,-176.461,6.815,148.222
C07018=1223.821,294.676,-66.374,-176.464,6.812,148.222
C07019=1223.826,294.428,-66.345,-176.466,6.809,148.222
C07020=1223.830,294.180,-66.315,-176.468,6.807,148.222
C07021=1223.835,293.931,-66.287,-176.471,6.805,148.222
C07022=1223.839,293.683,-66.257,-176.473,6.803,148.222
C07023=1223.844,293.435,-66.228,-176.476,6.800,148.222
C07024=1223.847,293.186,-66.200,-176.478,6.798,148.222
C07025=1223.851,292.938,-66.170,-176.480,6.796,148.222
C07026=1223.856,292.689,-66.142,-176.483,6.793,148.222
C07027=1223.861,292.442,-66.113,-176.485,6.791,148.223
C07028=1223.865,292.193,-66.083,-176.487,6.788,148.223
C07029=1223.869,291.945,-66.055,-176.490,6.786,148.223
C07030=1223.873,291.697,-66.026,-176.493,6.783,148.223
C07031=1223.878,291.448,-65.997,-176.495,6.781,148.223
C07032=1223.882,291.200,-65.968,-176.497,6.779,148.223
C07033=1223.886,290.952,-65.940,-176.500,6.776,148.223
C07034=1223.891,290.704,-65.910,-176.502,6.774,148.223
C07035=1223.895,290.455,-65.882,-176.504,6.772,148.223
C07036=1223.899,290.207,-65.852,-176.507,6.769,148.223
C07037=1223.904,289.959,-65.825,-176.509,6.767,148.224
C07038=1223.908,289.685,-65.793,-176.512,6.764,148.224
C07039=1223.913,289.410,-65.761,-176.515,6.762,148.224
C07040=1223.918,289.137,-65.729,-176.517,6.759,148.224
C07041=1223.923,288.862,-65.697,-176.519,6.757,148.224
C07042=1223.927,288.613,-65.668,-176.523,6.754,148.224
C07043=1223.932,288.366,-65.639,-176.525,6.752,148.224
C07044=1223.936,288.117,-65.611,-176.527,6.750,148.224
C07045=1223.940,287.868,-65.583,-176.530,6.747,148.225
C07046=1223.945,287.621,-65.553,-176.532,6.745,148.225
C07047=1223.949,287.372,-65.525,-176.534,6.742,148.225
C07048=1223.954,287.124,-65.497,-176.537,6.740,148.225
C07049=1223.958,286.876,-65.467,-176.539,6.737,148.225
C07050=1223.962,286.627,-65.439,-176.542,6.735,148.225
C07051=1223.967,286.379,-65.411,-176.544,6.733,148.225
C07052=1223.970,286.131,-65.382,-176.546,6.731,148.225
C07053=1223.975,285.882,-65.353,-176.549,6.728,148.225
C07054=1223.980,285.634,-65.325,-176.552,6.726,148.226
C07055=1223.983,285.385,-65.297,-176.554,6.724,148.226
C07056=1223.988,285.138,-65.268,-176.556,6.721,148.226
C07057=1223.992,284.889,-65.240,-176.559,6.719,148.226
C07058=1223.997,284.641,-65.211,-176.561,6.717,148.226
C07059=1224.002,284.392,-65.183,-176.563,6.715,148.226
C07060=1224.005,284.143,-65.154,-176.566,6.712,148.227
C07061=1224.010,283.896,-65.125,-176.568,6.710,148.227
C07062=1224.014,283.647,-65.097,-176.571,6.708,148.227
C07063=1224.019,283.399,-65.069,-176.573,6.706,148.227
C07064=1224.023,283.151,-65.041,-176.576,6.703,148.227
C07065=1224.028,282.902,-65.012,-176.578,6.701,148.227
C07066=1224.032,282.654,-64.984,-176.581,6.698,148.227
C07067=1224.036,282.405,-64.955,-176.583,6.696,148.227
C07068=1224.040,282.157,-64.928,-176.586,6.693,148.228
C07069=1224.045,281.909,-64.898,-176.588,6.691,148.228
C07070=1224.049,281.661,-64.870,-176.591,6.689,148.228
C07071=1224.053,281.412,-64.842,-176.593,6.687,148.228
C07072=1224.058,281.164,-64.814,-176.595,6.684,148.228
C07073=1224.062,280.915,-64.785,-176.598,6.682,148.228
C07074=1224.067,280.667,-64.757,-176.600,6.680,148.228
C07075=1224.071,280.418,-64.729,-176.603,6.678,148.229
C07076=1224.075,280.171,-64.701,-176.605,6.675,148.229
C07077=1224.079,279.922,-64.673,-176.607,6.673,148.229
C07078=1224.084,279.674,-64.644,-176.610,6.671,148.229
C07079=1224.088,279.425,-64.616,-176.612,6.669,148.229
C07080=1224.093,279.177,-64.588,-176.615,6.667,148.229
C07081=1224.097,278.929,-64.560,-176.617,6.664,148.229
C07082=1224.101,278.681,-64.532,-176.620,6.662,148.230
C07083=1224.106,278.431,-64.504,-176.622,6.660,148.230
C07084=1224.110,278.183,-64.476,-176.624,6.658,148.230
C07085=1224.115,277.934,-64.447,-176.627,6.655,148.230
C07086=1224.119,277.686,-64.420,-176.630,6.653,148.230
C07087=1224.123,277.438,-64.391,-176.632,6.651,148.231
C07088=1224.128,277.190,-64.363,-176.634,6.648,148.231
C07089=1224.132,276.942,-64.335,-176.637,6.646,148.231
C07090=1224.136,276.693,-64.307,-176.639,6.644,148.231
C07091=1224.142,276.444,-64.279,-176.642,6.642,148.231
C07092=1224.145,276.196,-64.251,-176.644,6.639,148.231
C07093=1224.150,275.948,-64.224,-176.647,6.638,148.232
C07094=1224.153,275.699,-64.195,-176.649,6.635,148.232
C07095=1224.158,275.451,-64.167,-176.652,6.632,148.232
C07096=1224.163,275.202,-64.140,-176.654,6.630,148.232
C07097=1224.167,274.954,-64.112,-176.656,6.628,148.232
C07098=1224.172,274.706,-64.083,-176.659,6.626,148.232
C07099=1224.176,274.457,-64.055,-176.662,6.623,148.232
C07100=1224.180,274.209,-64.028,-176.664,6.621,148.233
C07101=1224.184,273.960,-64.000,-176.666,6.619,148.233
C07102=1224.189,273.712,-63.972,-176.669,6.617,148.233
C07103=1224.194,273.464,-63.945,-176.671,6.615,148.233
C07104=1224.198,273.215,-63.917,-176.674,6.612,148.233
C07105=1224.202,272.967,-63.889,-176.676,6.610,148.233
C07106=1224.207,272.718,-63.861,-176.679,6.608,148.234
C07107=1224.211,272.470,-63.833,-176.681,6.606,148.234
C07108=1224.215,272.222,-63.805,-176.684,6.604,148.234
C07109=1224.220,271.973,-63.778,-176.686,6.601,148.234
C07110=1224.224,271.725,-63.750,-176.689,6.599,148.234
C07111=1224.228,271.477,-63.722,-176.691,6.597,148.234
C07112=1224.233,271.227,-63.694,-176.694,6.595,148.235
C07113=1224.237,270.980,-63.666,-176.696,6.593,148.235
C07114=1224.242,270.731,-63.639,-176.699,6.590,148.235
C07115=1224.246,270.483,-63.611,-176.702,6.588,148.235
C07116=1224.250,270.234,-63.584,-176.704,6.586,148.235
C07117=1224.255,269.986,-63.556,-176.706,6.584,148.236
C07118=1224.259,269.738,-63.529,-176.708,6.582,148.236
C07119=1224.264,269.489,-63.501,-176.711,6.580,148.236
C07120=1224.269,269.240,-63.473,-176.714,6.577,148.236
C07121=1224.273,268.992,-63.446,-176.716,6.575,148.236
C07122=1224.277,268.743,-63.418,-176.718,6.573,148.237
C07123=1224.281,268.495,-63.391,-176.721,6.571,148.237
C07124=1224.286,268.247,-63.363,-176.723,6.569,148.237
C07125=1224.290,267.998,-63.335,-176.726,6.567,148.237
C07126=1224.294,267.750,-63.308,-176.729,6.564,148.237
C07127=1224.299,267.502,-63.280,-176.731,6.562,148.238
C07128=1224.303,267.253,-63.253,-176.734,6.560,148.238
C07129=1224.307,267.004,-63.226,-176.736,6.558,148.238
C07130=1224.312,266.756,-63.198,-176.738,6.556,148.238
C07131=1224.316,266.508,-63.171,-176.740,6.554,148.238
C07132=1224.321,266.260,-63.143,-176.744,6.551,148.239
C07133=1224.325,266.011,-63.116,-176.746,6.549,148.239
C07134=1224.330,265.762,-63.089,-176.748,6.547,148.239
C07135=1224.334,265.514,-63.061,-176.751,6.545,148.239
C07136=1224.339,265.266,-63.034,-176.753,6.543,148.239
C07137=1224.343,265.017,-63.007,-176.756,6.541,148.240
C07138=1224.347,264.769,-62.979,-176.758,6.539,148.240
C07139=1224.352,264.520,-62.952,-176.761,6.536,148.240
C07140=1224.356,264.272,-62.925,-176.764,6.534,148.240
C07141=1224.361,264.023,-62.898,-176.766,6.532,148.240
C07142=1224.366,263.750,-62.867,-176.768,6.530,148.241
C07143=1224.370,263.478,-62.837,-176.771,6.527,148.241
C07144=1224.375,263.205,-62.807,-176.774,6.525,148.241
C07145=1224.380,262.933,-62.777,-176.777,6.523,148.241
C07146=1224.385,262.684,-62.750,-176.779,6.521,148.241
C07147=1224.389,262.436,-62.723,-176.781,6.518,148.242
C07148=1224.393,262.187,-62.696,-176.784,6.517,148.242
C07149=1224.398,261.938,-62.669,-176.787,6.515,148.242
C07150=1224.402,261.690,-62.641,-176.789,6.513,148.242
C07151=1224.406,261.442,-62.614,-176.791,6.511,148.243
C07152=1224.411,261.194,-62.587,-176.794,6.509,148.243
C07153=1224.415,260.945,-62.560,-176.797,6.506,148.243
C07154=1224.420,260.697,-62.533,-176.799,6.504,148.243
C07155=1224.424,260.447,-62.506,-176.801,6.502,148.243
C07156=1224.429,260.199,-62.479,-176.804,6.500,148.244
C07157=1224.434,259.950,-62.452,-176.807,6.498,148.244
C07158=1224.437,259.702,-62.425,-176.809,6.496,148.244
C07159=1224.442,259.454,-62.398,-176.811,6.494,148.244
C07160=1224.447,259.205,-62.371,-176.814,6.492,148.245
C07161=1224.451,258.957,-62.343,-176.817,6.489,148.245
C07162=1224.455,258.708,-62.316,-176.819,6.487,148.245
C07163=1224.459,258.460,-62.289,-176.822,6.485,148.245
C07164=1224.464,258.211,-62.262,-176.824,6.483,148.245
C07165=1224.468,257.963,-62.235,-176.827,6.481,148.246
C07166=1224.473,257.714,-62.209,-176.829,6.479,148.246
C07167=1224.477,257.466,-62.182,-176.831,6.477,148.246
C07168=1224.482,257.217,-62.155,-176.834,6.475,148.246
C07169=1224.487,256.969,-62.128,-176.837,6.473,148.247
C07170=1224.491,256.720,-62.101,-176.839,6.471,148.247
C07171=1224.495,256.472,-62.075,-176.842,6.468,148.247
C07172=1224.500,256.223,-62.048,-176.844,6.466,148.247
C07173=1224.504,255.974,-62.020,-176.847,6.464,148.247
C07174=1224.509,255.726,-61.993,-176.849,6.462,148.248
C07175=1224.512,255.478,-61.967,-176.852,6.460,148.248
C07176=1224.517,255.229,-61.940,-176.854,6.458,148.248
C07177=1224.522,254.980,-61.913,-176.857,6.456,148.248
C07178=1224.526,254.732,-61.887,-176.859,6.454,148.249
C07179=1224.531,254.483,-61.860,-176.861,6.452,148.249
C07180=1224.535,254.235,-61.833,-176.864,6.450,148.249
C07181=1224.539,253.987,-61.806,-176.866,6.448,148.249
C07182=1224.544,253.738,-61.779,-176.869,6.446,148.249
C07183=1224.548,253.489,-61.753,-176.872,6.444,148.250
C07184=1224.553,253.241,-61.726,-176.874,6.442,148.250
C07185=1224.557,252.992,-61.699,-176.877,6.439,148.250
C07186=1224.561,252.744,-61.673,-176.879,6.438,148.250
C07187=1224.566,252.495,-61.647,-176.882,6.436,148.251
C07188=1224.571,252.247,-61.620,-176.884,6.434,148.251
C07189=1224.575,251.998,-61.593,-176.886,6.432,148.251
C07190=1224.580,251.750,-61.566,-176.889,6.430,148.251
C07191=1224.584,251.501,-61.540,-176.892,6.428,148.252
C07192=1224.588,251.253,-61.513,-176.894,6.426,148.252
C07193=1224.592,251.004,-61.487,-176.896,6.424,148.252
C07194=1224.597,250.755,-61.460,-176.899,6.422,148.252
C07195=1224.602,250.507,-61.433,-176.902,6.420,148.253
C07196=1224.606,250.259,-61.407,-176.904,6.418,148.253
C07197=1224.611,250.009,-61.380,-176.906,6.416,148.253
C07198=1224.615,249.761,-61.354,-176.909,6.414,148.253
C07199=1224.620,249.512,-61.328,-176.912,6.411,148.253
C07200=1224.624,249.264,-61.301,-176.914,6.409,148.254
C07201=1224.628,249.015,-61.274,-176.917,6.407,148.254
C07202=1224.633,248.767,-61.248,-176.920,6.405,148.254
C07203=1224.638,248.519,-61.222,-176.922,6.403,148.254
C07204=1224.642,248.270,-61.196,-176.924,6.401,148.255
C07205=1224.647,248.022,-61.169,-176.927,6.399,148.255
C07206=1224.651,247.773,-61.143,-176.930,6.398,148.255
C07207=1224.656,247.524,-61.116,-176.932,6.395,148.255
C07208=1224.660,247.275,-61.090,-176.934,6.394,148.256
C07209=1224.664,247.027,-61.064,-176.937,6.392,148.256
C07210=1224.669,246.778,-61.038,-176.939,6.390,148.256
C07211=1224.673,246.530,-61.011,-176.942,6.388,148.256
C07212=1224.678,246.281,-60.985,-176.944,6.386,148.257
C07213=1224.681,246.033,-60.958,-176.947,6.384,148.257
C07214=1224.687,245.784,-60.932,-176.949,6.382,148.257
C07215=1224.691,245.536,-60.906,-176.952,6.380,148.258
C07216=1224.695,245.287,-60.880,-176.954,6.378,148.258
C07217=1224.700,245.038,-60.854,-176.957,6.376,148.258
C07218=1224.704,244.790,-60.827,-176.959,6.374,148.258
C07219=1224.709,244.541,-60.801,-176.962,6.372,148.259
C07220=1224.713,244.293,-60.774,-176.964,6.370,148.259
C07221=1224.717,244.044,-60.749,-176.967,6.368,148.259
C07222=1224.723,243.795,-60.723,-176.969,6.366,148.259
C07223=1224.727,243.547,-60.696,-176.972,6.364,148.260
C07224=1224.731,243.298,-60.670,-176.974,6.362,148.260
C07225=1224.736,243.049,-60.644,-176.977,6.360,148.260
C07226=1224.740,242.801,-60.618,-176.979,6.358,148.261
C07227=1224.744,242.552,-60.592,-176.982,6.357,148.261
C07228=1224.750,242.304,-60.566,-176.985,6.355,148.261
C07229=1224.753,242.056,-60.539,-176.987,6.353,148.261
C07230=1224.758,241.807,-60.514,-176.989,6.351,148.262
C07231=1224.762,241.558,-60.488,-176.992,6.349,148.262
C07232=1224.767,241.309,-60.462,-176.995,6.347,148.262
C07233=1224.771,241.062,-60.435,-176.997,6.345,148.262
C07234=1224.776,240.813,-60.410,-176.999,6.343,148.263
C07235=1224.781,240.564,-60.383,-177.002,6.341,148.263
C07236=1224.785,240.315,-60.358,-177.005,6.339,148.263
C07237=1224.789,240.066,-60.332,-177.007,6.337,148.264
C07238=1224.794,239.819,-60.306,-177.010,6.335,148.264
C07239=1224.798,239.569,-60.279,-177.012,6.333,148.264
C07240=1224.803,239.321,-60.254,-177.015,6.331,148.264
C07241=1224.807,239.072,-60.228,-177.017,6.329,148.265
C07242=1224.812,238.824,-60.203,-177.020,6.328,148.265
C07243=1224.816,238.575,-60.177,-177.022,6.326,148.265
C07244=1224.821,238.326,-60.150,-177.025,6.323,148.265
C07245=1224.825,238.077,-60.125,-177.027,6.322,148.266
C07246=1224.830,237.806,-60.096,-177.030,6.319,148.266
C07247=1224.835,237.535,-60.068,-177.033,6.317,148.266
C07248=1224.840,237.263,-60.041,-177.036,6.315,148.267
C07249=1224.845,236.992,-60.012,-177.038,6.313,148.267
C07250=1224.849,236.743,-59.986,-177.041,6.311,148.267
C07251=1224.854,236.495,-59.961,-177.043,6.310,148.267
C07252=1224.858,236.246,-59.935,-177.046,6.308,148.268
C07253=1224.863,235.997,-59.909,-177.049,6.306,148.268
C07254=1224.867,235.748,-59.883,-177.051,6.304,148.268
C07255=1224.872,235.500,-59.857,-177.053,6.302,148.269
C07256=1224.876,235.252,-59.832,-177.056,6.300,148.269
C07257=1224.880,235.003,-59.806,-177.059,6.298,148.269
C07258=1224.885,234.755,-59.781,-177.061,6.296,148.269
C07259=1224.889,234.506,-59.755,-177.064,6.294,148.270
C07260=1224.894,234.257,-59.729,-177.067,6.292,148.270
C07261=1224.898,234.009,-59.704,-177.069,6.290,148.270
C07262=1224.903,233.760,-59.678,-177.071,6.288,148.271
C07263=1224.907,233.511,-59.653,-177.074,6.286,148.271
C07264=1224.912,233.263,-59.628,-177.077,6.285,148.271
C07265=1224.916,233.014,-59.602,-177.079,6.283,148.271
C07266=1224.920,232.765,-59.576,-177.082,6.281,148.272
C07267=1224.926,232.517,-59.550,-177.084,6.279,148.272
C07268=1224.930,232.268,-59.524,-177.087,6.277,148.272
C07269=1224.934,232.019,-59.499,-177.089,6.275,148.273
C07270=1224.940,231.770,-59.474,-177.092,6.273,148.273
C07271=1224.944,231.521,-59.448,-177.094,6.271,148.273
C07272=1224.949,231.273,-59.423,-177.097,6.269,148.273
C07273=1224.952,231.025,-59.398,-177.099,6.268,148.274
C07274=1224.956,230.776,-59.372,-177.102,6.266,148.274
C07275=1224.961,230.527,-59.347,-177.104,6.265,148.275
C07276=1224.966,230.278,-59.321,-177.107,6.263,148.275
C07277=1224.970,230.030,-59.296,-177.109,6.261,148.275
C07278=1224.975,229.782,-59.270,-177.112,6.259,148.275
C07279=1224.979,229.532,-59.245,-177.114,6.257,148.276
C07280=1224.984,229.284,-59.220,-177.117,6.255,148.276
C07281=1224.988,229.035,-59.194,-177.120,6.253,148.276
C07282=1224.993,228.786,-59.169,-177.122,6.251,148.277
C07283=1224.998,228.538,-59.144,-177.125,6.249,148.277
C07284=1225.002,228.289,-59.118,-177.127,6.247,148.277
C07285=1225.007,228.040,-59.093,-177.130,6.246,148.277
C07286=1225.011,227.791,-59.068,-177.133,6.244,148.278
C07287=1225.015,227.544,-59.043,-177.135,6.242,148.278
C07288=1225.020,227.294,-59.018,-177.137,6.240,148.278
C07289=1225.025,227.046,-58.992,-177.140,6.239,148.279
C07290=1225.029,226.797,-58.967,-177.142,6.237,148.279
C07291=1225.034,226.549,-58.942,-177.145,6.235,148.279
C07292=1225.038,226.300,-58.916,-177.147,6.233,148.280
C07293=1225.043,226.050,-58.891,-177.150,6.231,148.280
C07294=1225.047,225.802,-58.866,-177.153,6.229,148.280
C07295=1225.051,225.553,-58.841,-177.155,6.227,148.281
C07296=1225.056,225.305,-58.816,-177.158,6.226,148.281
C07297=1225.060,225.056,-58.790,-177.161,6.224,148.281
C07298=1225.066,224.807,-58.765,-177.163,6.222,148.282
